      A     M      3.3;
      =     L      0.0;
      A     L      0.0;
      A     I    264.2;
      AN    I    264.3;
      =     M   2102.2;
      A     L      0.0;
      AN    I    264.2;
      A     I    264.3;
      =     M   2102.3;
NETWORK
TITLE =

      A     M      3.3;
      =     L      0.0;
      A     L      0.0;
      A     I    264.4;
      AN    I    264.5;
      =     M   2102.4;
      A     L      0.0;
      AN    I    264.4;
      A     I    264.5;
      =     M   2102.5;
NETWORK
TITLE =
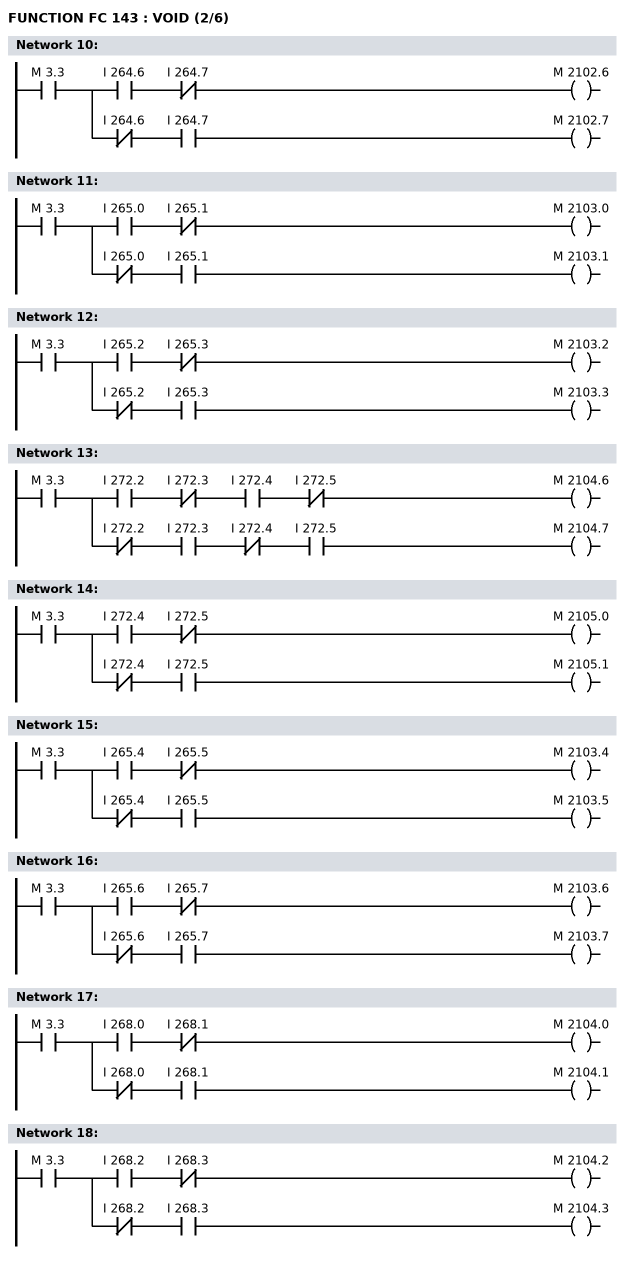

      A     M      3.3;
      =     L      0.0;
      A     L      0.0;
      A     I    264.6;
      AN    I    264.7;
      =     M   2102.6;
      A     L      0.0;
      AN    I    264.6;
      A     I    264.7;
      =     M   2102.7;
NETWORK
TITLE =

      A     M      3.3;
      =     L      0.0;
      A     L      0.0;
      A     I    265.0;
      AN    I    265.1;
      =     M   2103.0;
      A     L      0.0;
      AN    I    265.0;
      A     I    265.1;
      =     M   2103.1;
NETWORK
TITLE =

      A     M      3.3;
      =     L      0.0;
      A     L      0.0;
      A     I    265.2;
      AN    I    265.3;
      =     M   2103.2;
      A     L      0.0;
      AN    I    265.2;
      A     I    265.3;
      =     M   2103.3;
NETWORK
TITLE =

      A     M      3.3;
      =     L      0.0;
      A     L      0.0;
      A     I    272.2;
      AN    I    272.3;
      A     I    272.4;
      AN    I    272.5;
      =     M   2104.6;
      A     L      0.0;
      AN    I    272.2;
      A     I    272.3;
      AN    I    272.4;
      A     I    272.5;
      =     M   2104.7;
NETWORK
TITLE =

      A     M      3.3;
      =     L      0.0;
      A     L      0.0;
      A     I    272.4;
      AN    I    272.5;
      =     M   2105.0;
      A     L      0.0;
      AN    I    272.4;
      A     I    272.5;
      =     M   2105.1;
NETWORK
TITLE =

      A     M      3.3;
      =     L      0.0;
      A     L      0.0;
      A     I    265.4;
      AN    I    265.5;
      =     M   2103.4;
      A     L      0.0;
      AN    I    265.4;
      A     I    265.5;
      =     M   2103.5;
NETWORK
TITLE =

      A     M      3.3;
      =     L      0.0;
      A     L      0.0;
      A     I    265.6;
      AN    I    265.7;
      =     M   2103.6;
      A     L      0.0;
      AN    I    265.6;
      A     I    265.7;
      =     M   2103.7;
NETWORK
TITLE =

      A     M      3.3;
      =     L      0.0;
      A     L      0.0;
      A     I    268.0;
      AN    I    268.1;
      =     M   2104.0;
      A     L      0.0;
      AN    I    268.0;
      A     I    268.1;
      =     M   2104.1;
NETWORK
TITLE =

      A     M      3.3;
      =     L      0.0;
      A     L      0.0;
      A     I    268.2;
      AN    I    268.3;
      =     M   2104.2;
      A     L      0.0;
      AN    I    268.2;
      A     I    268.3;
      =     M   2104.3;
NETWORK
TITLE =
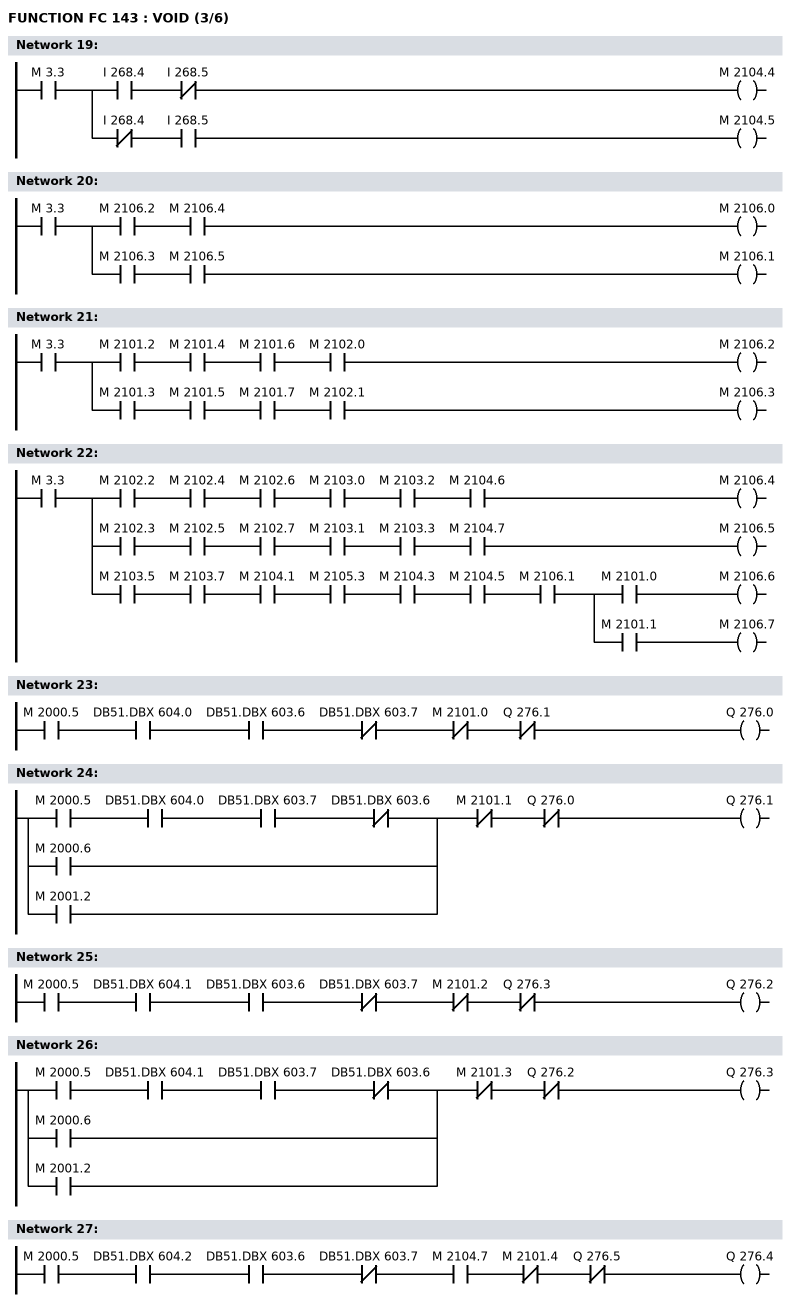

      A     M      3.3;
      =     L      0.0;
      A     L      0.0;
      A     I    268.4;
      AN    I    268.5;
      =     M   2104.4;
      A     L      0.0;
      AN    I    268.4;
      A     I    268.5;
      =     M   2104.5;
NETWORK
TITLE =

      A     M      3.3;
      =     L      0.0;
      A     L      0.0;
      A     M   2106.2;
      A     M   2106.4;
      =     M   2106.0;
      A     L      0.0;
      A     M   2106.3;
      A     M   2106.5;
      =     M   2106.1;
NETWORK
TITLE =

      A     M      3.3;
      =     L      0.0;
      A     L      0.0;
      A     M   2101.2;
      A     M   2101.4;
      A     M   2101.6;
      A     M   2102.0;
      =     M   2106.2;
      A     L      0.0;
      A     M   2101.3;
      A     M   2101.5;
      A     M   2101.7;
      A     M   2102.1;
      =     M   2106.3;
NETWORK
TITLE =

      A     M      3.3;
      =     L      0.0;
      A     L      0.0;
      A     M   2102.2;
      A     M   2102.4;
      A     M   2102.6;
      A     M   2103.0;
      A     M   2103.2;
      A     M   2104.6;
      =     M   2106.4;
      A     L      0.0;
      A     M   2102.3;
      A     M   2102.5;
      A     M   2102.7;
      A     M   2103.1;
      A     M   2103.3;
      A     M   2104.7;
      =     M   2106.5;
      A     L      0.0;
      A     M   2103.5;
      A     M   2103.7;
      A     M   2104.1;
      A     M   2105.3;
      A     M   2104.3;
      A     M   2104.5;
      A     M   2106.1;
      =     L      0.1;
      A     L      0.1;
      A     M   2101.0;
      =     M   2106.6;
      A     L      0.1;
      A     M   2101.1;
      =     M   2106.7;
NETWORK
TITLE =

      A     M   2000.5;
      A     DB51.DBX  604.0;
      A     DB51.DBX  603.6;
      AN    DB51.DBX  603.7;
      AN    M   2101.0;
      AN    Q    276.1;
      =     Q    276.0;
NETWORK
TITLE =

      A(    ;
      A     M   2000.5;
      A     DB51.DBX  604.0;
      A     DB51.DBX  603.7;
      AN    DB51.DBX  603.6;
      O     M   2000.6;
      O     M   2001.2;
      )     ;
      AN    M   2101.1;
      AN    Q    276.0;
      =     Q    276.1;
NETWORK
TITLE =

      A     M   2000.5;
      A     DB51.DBX  604.1;
      A     DB51.DBX  603.6;
      AN    DB51.DBX  603.7;
      AN    M   2101.2;
      AN    Q    276.3;
      =     Q    276.2;
NETWORK
TITLE =

      A(    ;
      A     M   2000.5;
      A     DB51.DBX  604.1;
      A     DB51.DBX  603.7;
      AN    DB51.DBX  603.6;
      O     M   2000.6;
      O     M   2001.2;
      )     ;
      AN    M   2101.3;
      AN    Q    276.2;
      =     Q    276.3;
NETWORK
TITLE =

      A     M   2000.5;
      A     DB51.DBX  604.2;
      A     DB51.DBX  603.6;
      AN    DB51.DBX  603.7;
      A     M   2104.7;
      AN    M   2101.4;
      AN    Q    276.5;
      =     Q    276.4;
NETWORK
TITLE =
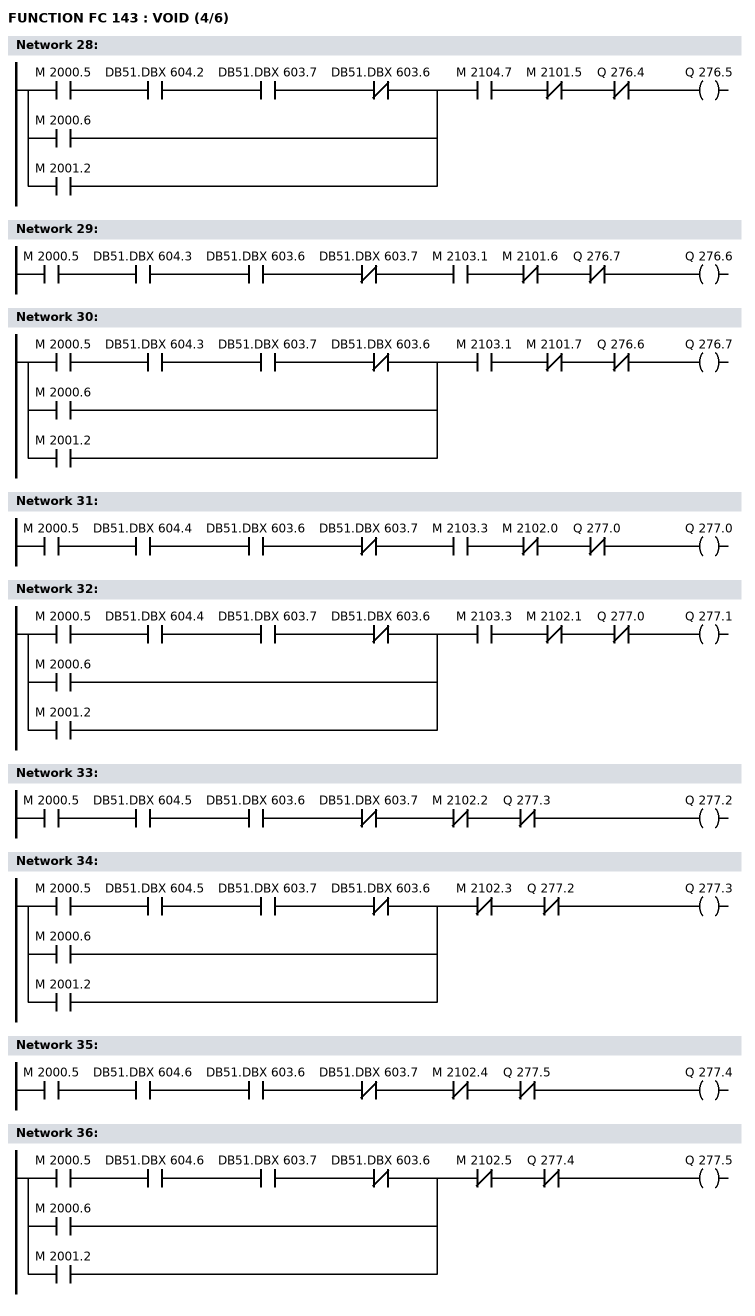

      A(    ;
      A     M   2000.5;
      A     DB51.DBX  604.2;
      A     DB51.DBX  603.7;
      AN    DB51.DBX  603.6;
      O     M   2000.6;
      O     M   2001.2;
      )     ;
      A     M   2104.7;
      AN    M   2101.5;
      AN    Q    276.4;
      =     Q    276.5;
NETWORK
TITLE =

      A     M   2000.5;
      A     DB51.DBX  604.3;
      A     DB51.DBX  603.6;
      AN    DB51.DBX  603.7;
      A     M   2103.1;
      AN    M   2101.6;
      AN    Q    276.7;
      =     Q    276.6;
NETWORK
TITLE =

      A(    ;
      A     M   2000.5;
      A     DB51.DBX  604.3;
      A     DB51.DBX  603.7;
      AN    DB51.DBX  603.6;
      O     M   2000.6;
      O     M   2001.2;
      )     ;
      A     M   2103.1;
      AN    M   2101.7;
      AN    Q    276.6;
      =     Q    276.7;
NETWORK
TITLE =

      A     M   2000.5;
      A     DB51.DBX  604.4;
      A     DB51.DBX  603.6;
      AN    DB51.DBX  603.7;
      A     M   2103.3;
      AN    M   2102.0;
      AN    Q    277.0;
      =     Q    277.0;
NETWORK
TITLE =

      A(    ;
      A     M   2000.5;
      A     DB51.DBX  604.4;
      A     DB51.DBX  603.7;
      AN    DB51.DBX  603.6;
      O     M   2000.6;
      O     M   2001.2;
      )     ;
      A     M   2103.3;
      AN    M   2102.1;
      AN    Q    277.0;
      =     Q    277.1;
NETWORK
TITLE =

      A     M   2000.5;
      A     DB51.DBX  604.5;
      A     DB51.DBX  603.6;
      AN    DB51.DBX  603.7;
      AN    M   2102.2;
      AN    Q    277.3;
      =     Q    277.2;
NETWORK
TITLE =

      A(    ;
      A     M   2000.5;
      A     DB51.DBX  604.5;
      A     DB51.DBX  603.7;
      AN    DB51.DBX  603.6;
      O     M   2000.6;
      O     M   2001.2;
      )     ;
      AN    M   2102.3;
      AN    Q    277.2;
      =     Q    277.3;
NETWORK
TITLE =

      A     M   2000.5;
      A     DB51.DBX  604.6;
      A     DB51.DBX  603.6;
      AN    DB51.DBX  603.7;
      AN    M   2102.4;
      AN    Q    277.5;
      =     Q    277.4;
NETWORK
TITLE =

      A(    ;
      A     M   2000.5;
      A     DB51.DBX  604.6;
      A     DB51.DBX  603.7;
      AN    DB51.DBX  603.6;
      O     M   2000.6;
      O     M   2001.2;
      )     ;
      AN    M   2102.5;
      AN    Q    277.4;
      =     Q    277.5;
NETWORK
TITLE =
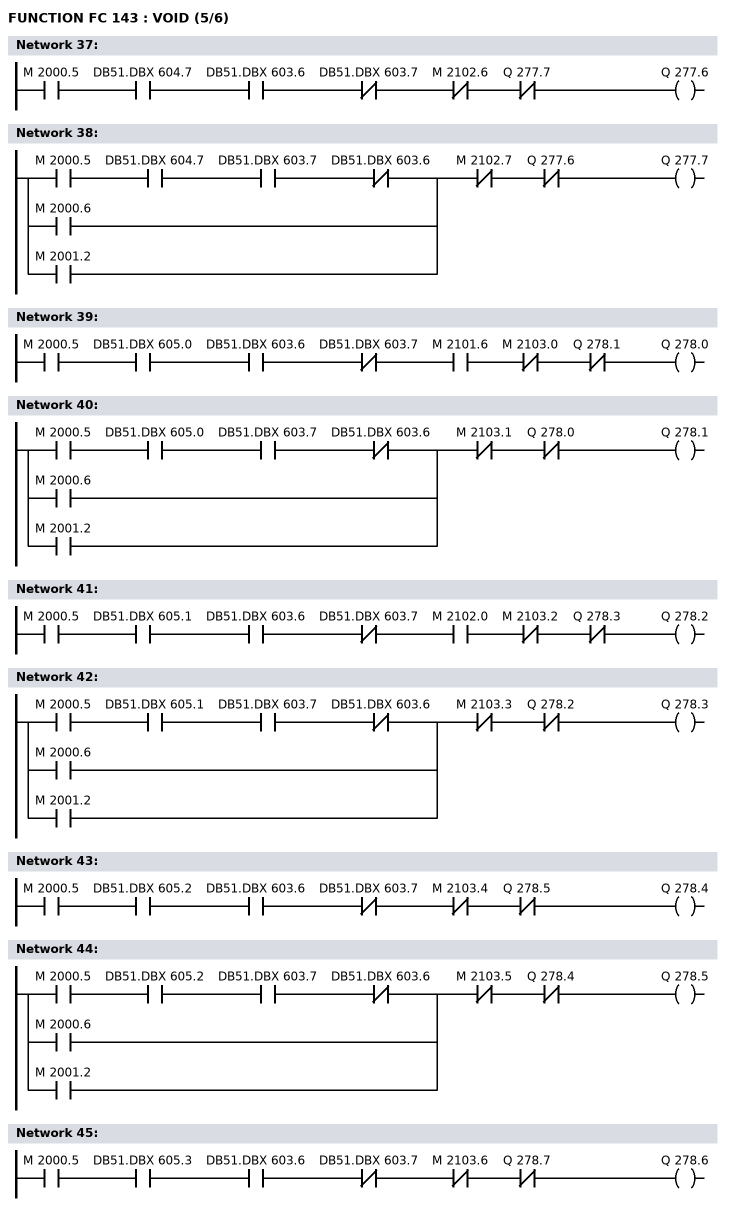

      A     M   2000.5;
      A     DB51.DBX  604.7;
      A     DB51.DBX  603.6;
      AN    DB51.DBX  603.7;
      AN    M   2102.6;
      AN    Q    277.7;
      =     Q    277.6;
NETWORK
TITLE =

      A(    ;
      A     M   2000.5;
      A     DB51.DBX  604.7;
      A     DB51.DBX  603.7;
      AN    DB51.DBX  603.6;
      O     M   2000.6;
      O     M   2001.2;
      )     ;
      AN    M   2102.7;
      AN    Q    277.6;
      =     Q    277.7;
NETWORK
TITLE =

      A     M   2000.5;
      A     DB51.DBX  605.0;
      A     DB51.DBX  603.6;
      AN    DB51.DBX  603.7;
      A     M   2101.6;
      AN    M   2103.0;
      AN    Q    278.1;
      =     Q    278.0;
NETWORK
TITLE =

      A(    ;
      A     M   2000.5;
      A     DB51.DBX  605.0;
      A     DB51.DBX  603.7;
      AN    DB51.DBX  603.6;
      O     M   2000.6;
      O     M   2001.2;
      )     ;
      AN    M   2103.1;
      AN    Q    278.0;
      =     Q    278.1;
NETWORK
TITLE =

      A     M   2000.5;
      A     DB51.DBX  605.1;
      A     DB51.DBX  603.6;
      AN    DB51.DBX  603.7;
      A     M   2102.0;
      AN    M   2103.2;
      AN    Q    278.3;
      =     Q    278.2;
NETWORK
TITLE =

      A(    ;
      A     M   2000.5;
      A     DB51.DBX  605.1;
      A     DB51.DBX  603.7;
      AN    DB51.DBX  603.6;
      O     M   2000.6;
      O     M   2001.2;
      )     ;
      AN    M   2103.3;
      AN    Q    278.2;
      =     Q    278.3;
NETWORK
TITLE =

      A     M   2000.5;
      A     DB51.DBX  605.2;
      A     DB51.DBX  603.6;
      AN    DB51.DBX  603.7;
      AN    M   2103.4;
      AN    Q    278.5;
      =     Q    278.4;
NETWORK
TITLE =

      A(    ;
      A     M   2000.5;
      A     DB51.DBX  605.2;
      A     DB51.DBX  603.7;
      AN    DB51.DBX  603.6;
      O     M   2000.6;
      O     M   2001.2;
      )     ;
      AN    M   2103.5;
      AN    Q    278.4;
      =     Q    278.5;
NETWORK
TITLE =

      A     M   2000.5;
      A     DB51.DBX  605.3;
      A     DB51.DBX  603.6;
      AN    DB51.DBX  603.7;
      AN    M   2103.6;
      AN    Q    278.7;
      =     Q    278.6;
NETWORK
TITLE =
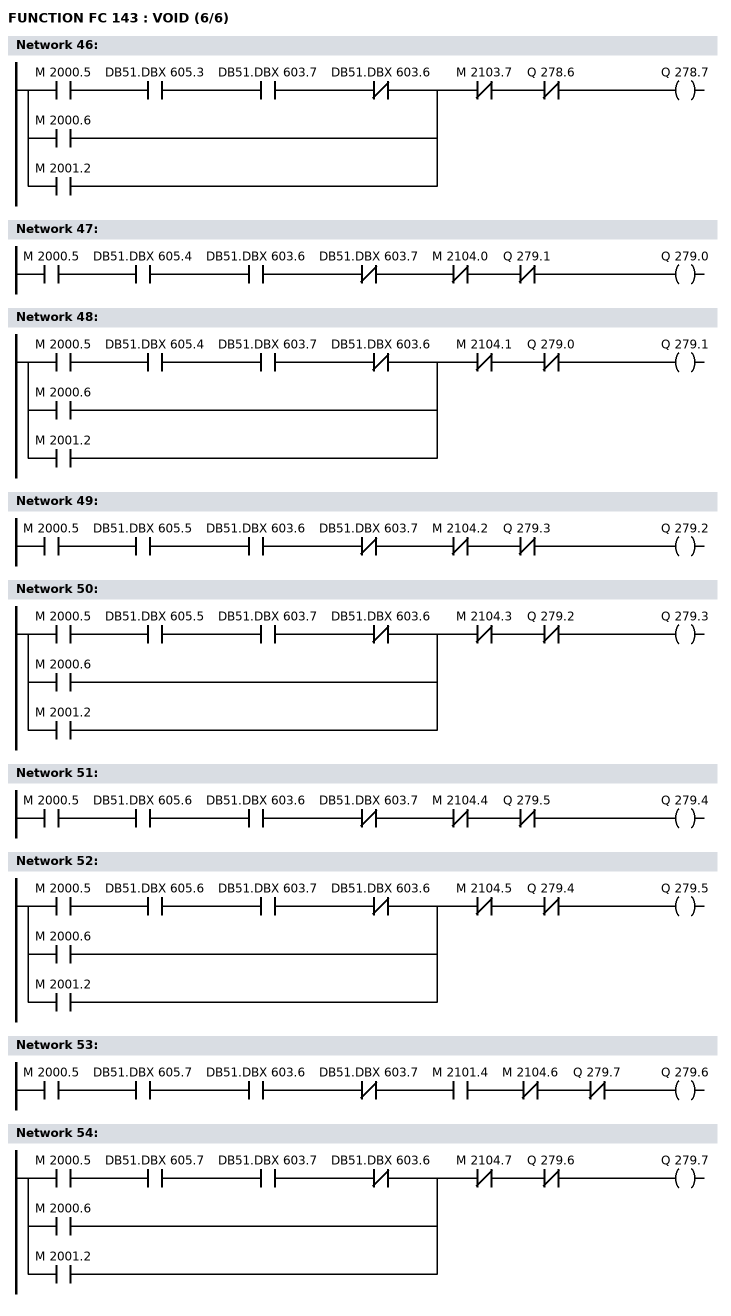

      A(    ;
      A     M   2000.5;
      A     DB51.DBX  605.3;
      A     DB51.DBX  603.7;
      AN    DB51.DBX  603.6;
      O     M   2000.6;
      O     M   2001.2;
      )     ;
      AN    M   2103.7;
      AN    Q    278.6;
      =     Q    278.7;
NETWORK
TITLE =

      A     M   2000.5;
      A     DB51.DBX  605.4;
      A     DB51.DBX  603.6;
      AN    DB51.DBX  603.7;
      AN    M   2104.0;
      AN    Q    279.1;
      =     Q    279.0;
NETWORK
TITLE =

      A(    ;
      A     M   2000.5;
      A     DB51.DBX  605.4;
      A     DB51.DBX  603.7;
      AN    DB51.DBX  603.6;
      O     M   2000.6;
      O     M   2001.2;
      )     ;
      AN    M   2104.1;
      AN    Q    279.0;
      =     Q    279.1;
NETWORK
TITLE =

      A     M   2000.5;
      A     DB51.DBX  605.5;
      A     DB51.DBX  603.6;
      AN    DB51.DBX  603.7;
      AN    M   2104.2;
      AN    Q    279.3;
      =     Q    279.2;
NETWORK
TITLE =

      A(    ;
      A     M   2000.5;
      A     DB51.DBX  605.5;
      A     DB51.DBX  603.7;
      AN    DB51.DBX  603.6;
      O     M   2000.6;
      O     M   2001.2;
      )     ;
      AN    M   2104.3;
      AN    Q    279.2;
      =     Q    279.3;
NETWORK
TITLE =

      A     M   2000.5;
      A     DB51.DBX  605.6;
      A     DB51.DBX  603.6;
      AN    DB51.DBX  603.7;
      AN    M   2104.4;
      AN    Q    279.5;
      =     Q    279.4;
NETWORK
TITLE =

      A(    ;
      A     M   2000.5;
      A     DB51.DBX  605.6;
      A     DB51.DBX  603.7;
      AN    DB51.DBX  603.6;
      O     M   2000.6;
      O     M   2001.2;
      )     ;
      AN    M   2104.5;
      AN    Q    279.4;
      =     Q    279.5;
NETWORK
TITLE =

      A     M   2000.5;
      A     DB51.DBX  605.7;
      A     DB51.DBX  603.6;
      AN    DB51.DBX  603.7;
      A     M   2101.4;
      AN    M   2104.6;
      AN    Q    279.7;
      =     Q    279.6;
NETWORK
TITLE =

      A(    ;
      A     M   2000.5;
      A     DB51.DBX  605.7;
      A     DB51.DBX  603.7;
      AN    DB51.DBX  603.6;
      O     M   2000.6;
      O     M   2001.2;
      )     ;
      AN    M   2104.7;
      AN    Q    279.6;
      =     Q    279.7;
END_FUNCTION

FUNCTION_BLOCK FB 144
TITLE =
VERSION : 0.1


VAR
  S708_TL_DC_PIN : FB 426;
  S708_TL_DC_LATCH1 : FB 426;
  S708_TL_DC_LATCH2 : FB 426;
  S708_TL_DC_1ST_CLAMP1 : FB 426;
  S708_TL_DC_1ST_CLAMP2 : FB 426;
  S708_TL_DC_1ST_CLAMP3 : FB 426;
  S708_TL_DC_2ND_CLAMP1 : FB 426;
  S708_TL_DC_2ND_CLAMP2 : FB 426;
  S708_TL_DC_U261 : FB 426;
  S708_TL_DC_U261_CLAMP : FB 426;
  S708_TL_DC_U269 : FB 426;
  S708_TL_DC_U269_CLAMP : FB 426;
  S708_TL_DC_3RD_CLAMP : FB 426;
  S708_TL_DC_U262_1_UP_DN : FB 426;
  S708_TL_DC_U262_1 : FB 426;
  S708_TL_DC_U262_1_CLAMP : FB 426;
  S708_TL_DC_U261_2_CLAMP : FB 426;
END_VAR
BEGIN
NETWORK
TITLE =
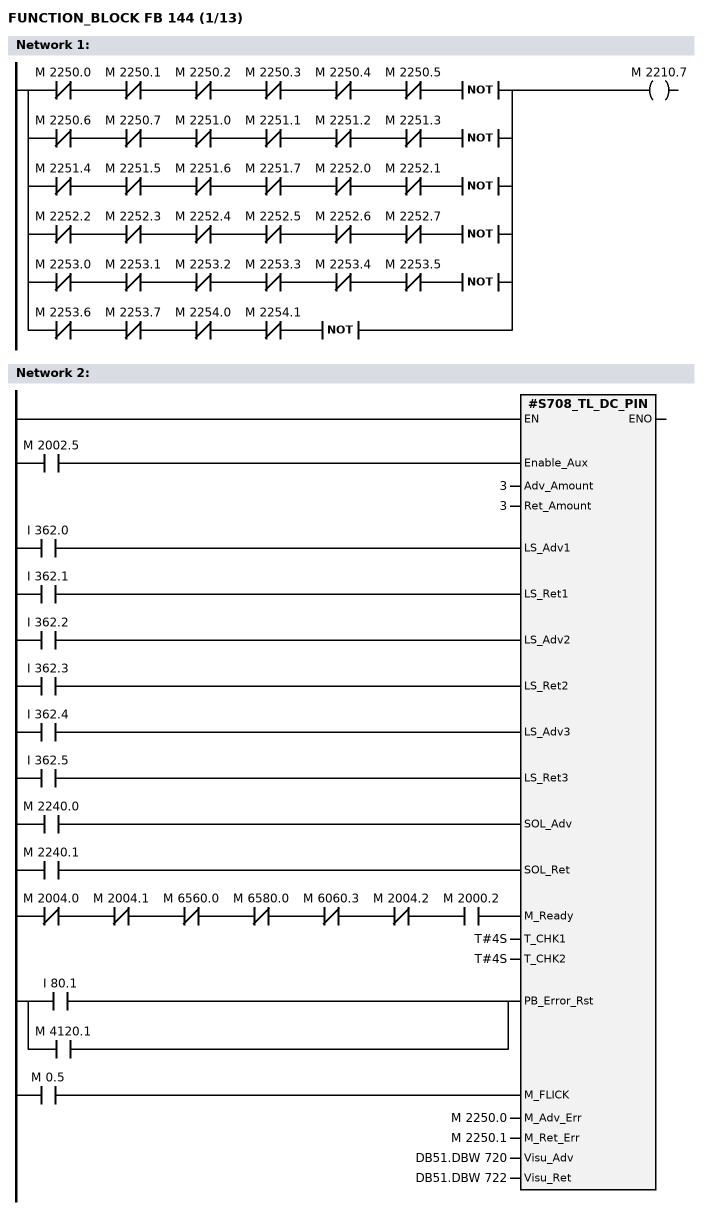

      AN    M   2250.0;
      AN    M   2250.1;
      AN    M   2250.2;
      AN    M   2250.3;
      AN    M   2250.4;
      AN    M   2250.5;
      NOT   ;
      O(    ;
      AN    M   2250.6;
      AN    M   2250.7;
      AN    M   2251.0;
      AN    M   2251.1;
      AN    M   2251.2;
      AN    M   2251.3;
      NOT   ;
      )     ;
      O(    ;
      AN    M   2251.4;
      AN    M   2251.5;
      AN    M   2251.6;
      AN    M   2251.7;
      AN    M   2252.0;
      AN    M   2252.1;
      NOT   ;
      )     ;
      O(    ;
      AN    M   2252.2;
      AN    M   2252.3;
      AN    M   2252.4;
      AN    M   2252.5;
      AN    M   2252.6;
      AN    M   2252.7;
      NOT   ;
      )     ;
      O(    ;
      AN    M   2253.0;
      AN    M   2253.1;
      AN    M   2253.2;
      AN    M   2253.3;
      AN    M   2253.4;
      AN    M   2253.5;
      NOT   ;
      )     ;
      O(    ;
      AN    M   2253.6;
      AN    M   2253.7;
      AN    M   2254.0;
      AN    M   2254.1;
      NOT   ;
      )     ;
      =     M   2210.7;
NETWORK
TITLE =

      A     M   2002.5;
      =     L      0.0;
      BLD   103;
      A     I    362.0;
      =     L      0.1;
      BLD   103;
      A     I    362.1;
      =     L      0.2;
      BLD   103;
      A     I    362.2;
      =     L      0.3;
      BLD   103;
      A     I    362.3;
      =     L      0.4;
      BLD   103;
      A     I    362.4;
      =     L      0.5;
      BLD   103;
      A     I    362.5;
      =     L      0.6;
      BLD   103;
      A     M   2240.0;
      =     L      2.1;
      BLD   103;
      A     M   2240.1;
      =     L      2.2;
      BLD   103;
      AN    M   2004.0;
      AN    M   2004.1;
      AN    M   6560.0;
      AN    M   6580.0;
      AN    M   6060.3;
      AN    M   2004.2;
      A     M   2000.2;
      =     L      2.3;
      BLD   103;
      A(    ;
      O     I     80.1;
      O     M   4120.1;
      )     ;
      =     L      2.5;
      BLD   103;
      A     M      0.5;
      =     L      2.6;
      BLD   103;
      CALL #S708_TL_DC_PIN (
           Enable_Aux               := L      0.0,
           Adv_Amount               := 3,
           Ret_Amount               := 3,
           LS_Adv1                  := L      0.1,
           LS_Ret1                  := L      0.2,
           LS_Adv2                  := L      0.3,
           LS_Ret2                  := L      0.4,
           LS_Adv3                  := L      0.5,
           LS_Ret3                  := L      0.6,
           SOL_Adv                  := L      2.1,
           SOL_Ret                  := L      2.2,
           M_Ready                  := L      2.3,
           T_CHK1                   := T#4S,
           T_CHK2                   := T#4S,
           PB_Error_Rst             := L      2.5,
           M_FLICK                  := L      2.6,
           M_Adv_Err                := M   2250.0,
           M_Ret_Err                := M   2250.1,
           Visu_Adv                 := DB51.DBW  720,
           Visu_Ret                 := DB51.DBW  722);
      NOP   0;
NETWORK
TITLE =
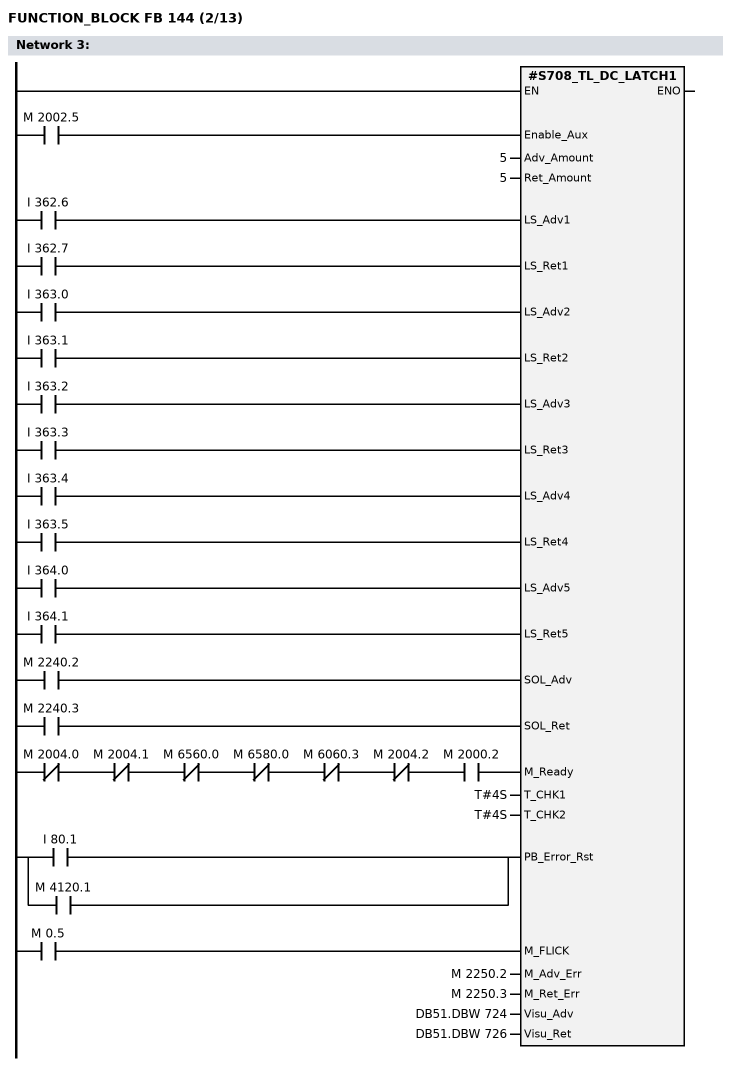

      A     M   2002.5;
      =     L      0.0;
      BLD   103;
      A     I    362.6;
      =     L      0.1;
      BLD   103;
      A     I    362.7;
      =     L      0.2;
      BLD   103;
      A     I    363.0;
      =     L      0.3;
      BLD   103;
      A     I    363.1;
      =     L      0.4;
      BLD   103;
      A     I    363.2;
      =     L      0.5;
      BLD   103;
      A     I    363.3;
      =     L      0.6;
      BLD   103;
      A     I    363.4;
      =     L      0.7;
      BLD   103;
      A     I    363.5;
      =     L      1.0;
      BLD   103;
      A     I    364.0;
      =     L      1.1;
      BLD   103;
      A     I    364.1;
      =     L      1.2;
      BLD   103;
      A     M   2240.2;
      =     L      2.1;
      BLD   103;
      A     M   2240.3;
      =     L      2.2;
      BLD   103;
      AN    M   2004.0;
      AN    M   2004.1;
      AN    M   6560.0;
      AN    M   6580.0;
      AN    M   6060.3;
      AN    M   2004.2;
      A     M   2000.2;
      =     L      2.3;
      BLD   103;
      A(    ;
      O     I     80.1;
      O     M   4120.1;
      )     ;
      =     L      2.5;
      BLD   103;
      A     M      0.5;
      =     L      2.6;
      BLD   103;
      CALL #S708_TL_DC_LATCH1 (
           Enable_Aux               := L      0.0,
           Adv_Amount               := 5,
           Ret_Amount               := 5,
           LS_Adv1                  := L      0.1,
           LS_Ret1                  := L      0.2,
           LS_Adv2                  := L      0.3,
           LS_Ret2                  := L      0.4,
           LS_Adv3                  := L      0.5,
           LS_Ret3                  := L      0.6,
           LS_Adv4                  := L      0.7,
           LS_Ret4                  := L      1.0,
           LS_Adv5                  := L      1.1,
           LS_Ret5                  := L      1.2,
           SOL_Adv                  := L      2.1,
           SOL_Ret                  := L      2.2,
           M_Ready                  := L      2.3,
           T_CHK1                   := T#4S,
           T_CHK2                   := T#4S,
           PB_Error_Rst             := L      2.5,
           M_FLICK                  := L      2.6,
           M_Adv_Err                := M   2250.2,
           M_Ret_Err                := M   2250.3,
           Visu_Adv                 := DB51.DBW  724,
           Visu_Ret                 := DB51.DBW  726);
      NOP   0;
NETWORK
TITLE =
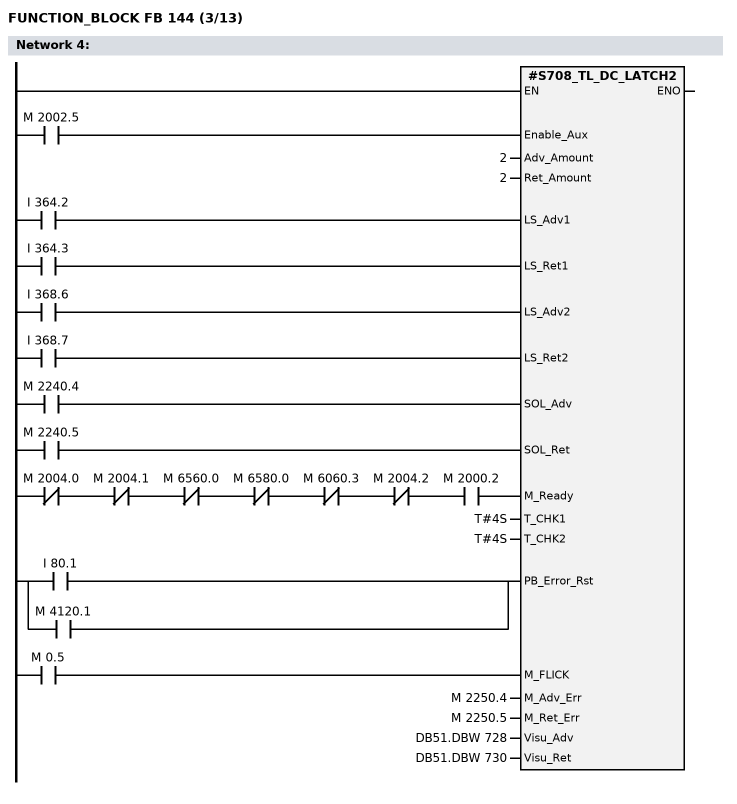

      A     M   2002.5;
      =     L      0.0;
      BLD   103;
      A     I    364.2;
      =     L      0.1;
      BLD   103;
      A     I    364.3;
      =     L      0.2;
      BLD   103;
      A     I    368.6;
      =     L      0.3;
      BLD   103;
      A     I    368.7;
      =     L      0.4;
      BLD   103;
      A     M   2240.4;
      =     L      2.1;
      BLD   103;
      A     M   2240.5;
      =     L      2.2;
      BLD   103;
      AN    M   2004.0;
      AN    M   2004.1;
      AN    M   6560.0;
      AN    M   6580.0;
      AN    M   6060.3;
      AN    M   2004.2;
      A     M   2000.2;
      =     L      2.3;
      BLD   103;
      A(    ;
      O     I     80.1;
      O     M   4120.1;
      )     ;
      =     L      2.5;
      BLD   103;
      A     M      0.5;
      =     L      2.6;
      BLD   103;
      CALL #S708_TL_DC_LATCH2 (
           Enable_Aux               := L      0.0,
           Adv_Amount               := 2,
           Ret_Amount               := 2,
           LS_Adv1                  := L      0.1,
           LS_Ret1                  := L      0.2,
           LS_Adv2                  := L      0.3,
           LS_Ret2                  := L      0.4,
           SOL_Adv                  := L      2.1,
           SOL_Ret                  := L      2.2,
           M_Ready                  := L      2.3,
           T_CHK1                   := T#4S,
           T_CHK2                   := T#4S,
           PB_Error_Rst             := L      2.5,
           M_FLICK                  := L      2.6,
           M_Adv_Err                := M   2250.4,
           M_Ret_Err                := M   2250.5,
           Visu_Adv                 := DB51.DBW  728,
           Visu_Ret                 := DB51.DBW  730);
      NOP   0;
NETWORK
TITLE =
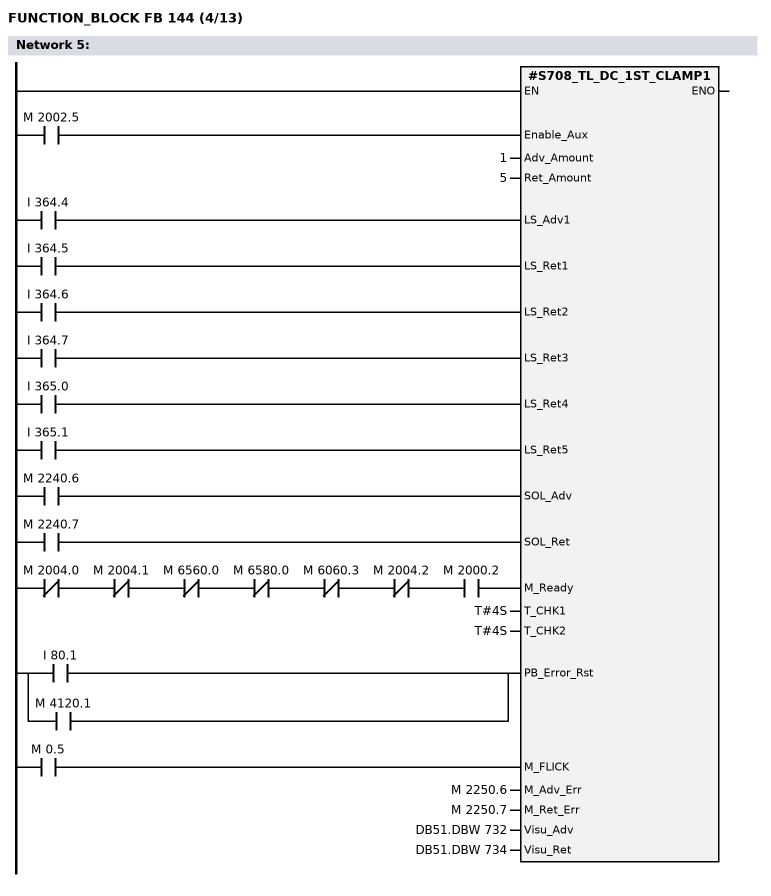

      A     M   2002.5;
      =     L      0.0;
      BLD   103;
      A     I    364.4;
      =     L      0.1;
      BLD   103;
      A     I    364.5;
      =     L      0.2;
      BLD   103;
      A     I    364.6;
      =     L      0.4;
      BLD   103;
      A     I    364.7;
      =     L      0.6;
      BLD   103;
      A     I    365.0;
      =     L      1.0;
      BLD   103;
      A     I    365.1;
      =     L      1.2;
      BLD   103;
      A     M   2240.6;
      =     L      2.1;
      BLD   103;
      A     M   2240.7;
      =     L      2.2;
      BLD   103;
      AN    M   2004.0;
      AN    M   2004.1;
      AN    M   6560.0;
      AN    M   6580.0;
      AN    M   6060.3;
      AN    M   2004.2;
      A     M   2000.2;
      =     L      2.3;
      BLD   103;
      A(    ;
      O     I     80.1;
      O     M   4120.1;
      )     ;
      =     L      2.5;
      BLD   103;
      A     M      0.5;
      =     L      2.6;
      BLD   103;
      CALL #S708_TL_DC_1ST_CLAMP1 (
           Enable_Aux               := L      0.0,
           Adv_Amount               := 1,
           Ret_Amount               := 5,
           LS_Adv1                  := L      0.1,
           LS_Ret1                  := L      0.2,
           LS_Ret2                  := L      0.4,
           LS_Ret3                  := L      0.6,
           LS_Ret4                  := L      1.0,
           LS_Ret5                  := L      1.2,
           SOL_Adv                  := L      2.1,
           SOL_Ret                  := L      2.2,
           M_Ready                  := L      2.3,
           T_CHK1                   := T#4S,
           T_CHK2                   := T#4S,
           PB_Error_Rst             := L      2.5,
           M_FLICK                  := L      2.6,
           M_Adv_Err                := M   2250.6,
           M_Ret_Err                := M   2250.7,
           Visu_Adv                 := DB51.DBW  732,
           Visu_Ret                 := DB51.DBW  734);
      NOP   0;
NETWORK
TITLE =
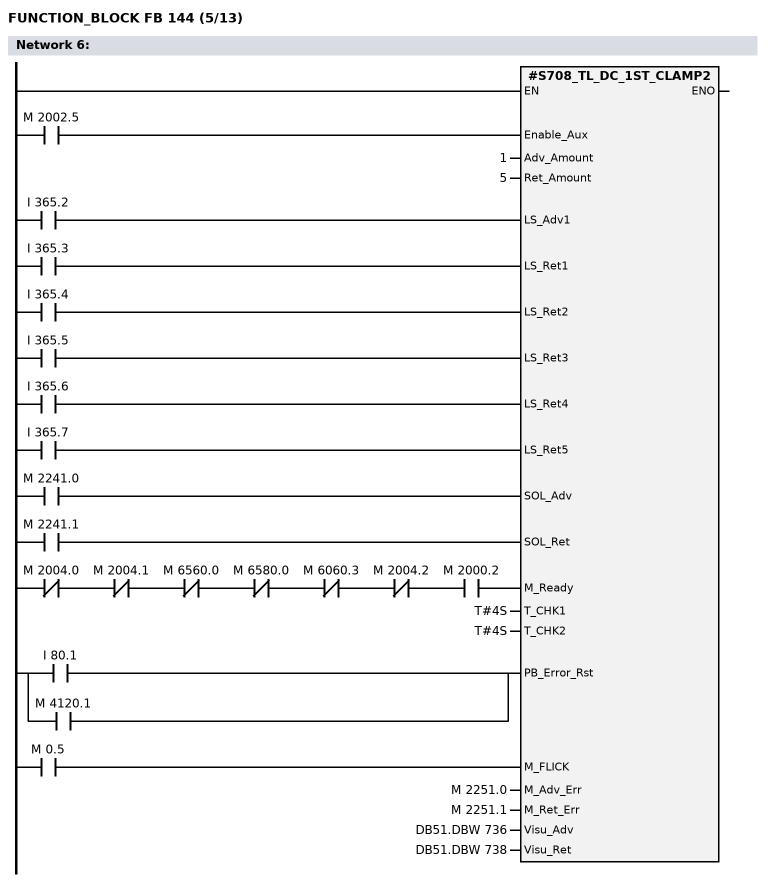

      A     M   2002.5;
      =     L      0.0;
      BLD   103;
      A     I    365.2;
      =     L      0.1;
      BLD   103;
      A     I    365.3;
      =     L      0.2;
      BLD   103;
      A     I    365.4;
      =     L      0.4;
      BLD   103;
      A     I    365.5;
      =     L      0.6;
      BLD   103;
      A     I    365.6;
      =     L      1.0;
      BLD   103;
      A     I    365.7;
      =     L      1.2;
      BLD   103;
      A     M   2241.0;
      =     L      2.1;
      BLD   103;
      A     M   2241.1;
      =     L      2.2;
      BLD   103;
      AN    M   2004.0;
      AN    M   2004.1;
      AN    M   6560.0;
      AN    M   6580.0;
      AN    M   6060.3;
      AN    M   2004.2;
      A     M   2000.2;
      =     L      2.3;
      BLD   103;
      A(    ;
      O     I     80.1;
      O     M   4120.1;
      )     ;
      =     L      2.5;
      BLD   103;
      A     M      0.5;
      =     L      2.6;
      BLD   103;
      CALL #S708_TL_DC_1ST_CLAMP2 (
           Enable_Aux               := L      0.0,
           Adv_Amount               := 1,
           Ret_Amount               := 5,
           LS_Adv1                  := L      0.1,
           LS_Ret1                  := L      0.2,
           LS_Ret2                  := L      0.4,
           LS_Ret3                  := L      0.6,
           LS_Ret4                  := L      1.0,
           LS_Ret5                  := L      1.2,
           SOL_Adv                  := L      2.1,
           SOL_Ret                  := L      2.2,
           M_Ready                  := L      2.3,
           T_CHK1                   := T#4S,
           T_CHK2                   := T#4S,
           PB_Error_Rst             := L      2.5,
           M_FLICK                  := L      2.6,
           M_Adv_Err                := M   2251.0,
           M_Ret_Err                := M   2251.1,
           Visu_Adv                 := DB51.DBW  736,
           Visu_Ret                 := DB51.DBW  738);
      NOP   0;
NETWORK
TITLE =
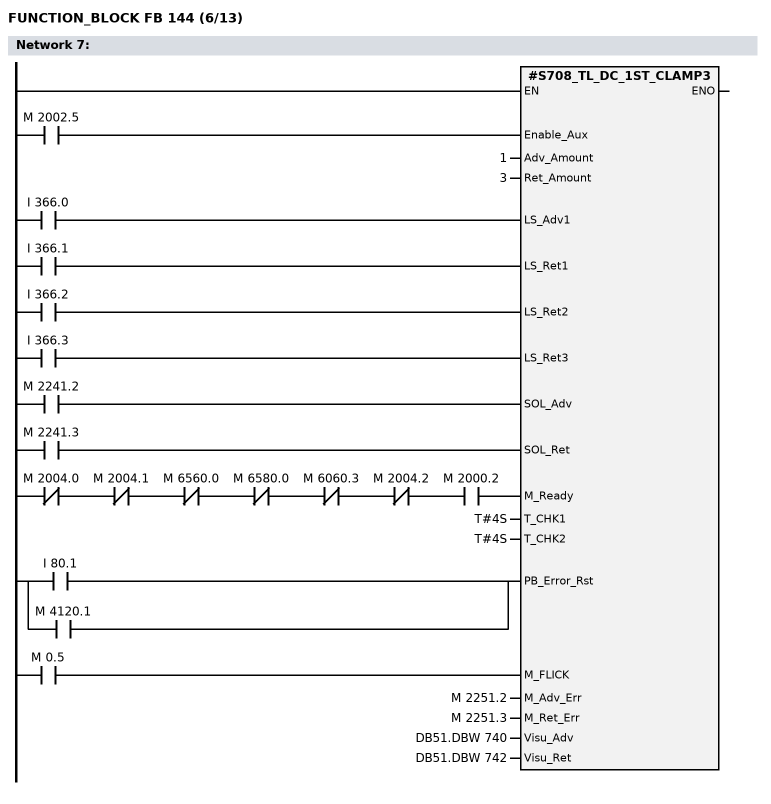

      A     M   2002.5;
      =     L      0.0;
      BLD   103;
      A     I    366.0;
      =     L      0.1;
      BLD   103;
      A     I    366.1;
      =     L      0.2;
      BLD   103;
      A     I    366.2;
      =     L      0.4;
      BLD   103;
      A     I    366.3;
      =     L      0.6;
      BLD   103;
      A     M   2241.2;
      =     L      2.1;
      BLD   103;
      A     M   2241.3;
      =     L      2.2;
      BLD   103;
      AN    M   2004.0;
      AN    M   2004.1;
      AN    M   6560.0;
      AN    M   6580.0;
      AN    M   6060.3;
      AN    M   2004.2;
      A     M   2000.2;
      =     L      2.3;
      BLD   103;
      A(    ;
      O     I     80.1;
      O     M   4120.1;
      )     ;
      =     L      2.5;
      BLD   103;
      A     M      0.5;
      =     L      2.6;
      BLD   103;
      CALL #S708_TL_DC_1ST_CLAMP3 (
           Enable_Aux               := L      0.0,
           Adv_Amount               := 1,
           Ret_Amount               := 3,
           LS_Adv1                  := L      0.1,
           LS_Ret1                  := L      0.2,
           LS_Ret2                  := L      0.4,
           LS_Ret3                  := L      0.6,
           SOL_Adv                  := L      2.1,
           SOL_Ret                  := L      2.2,
           M_Ready                  := L      2.3,
           T_CHK1                   := T#4S,
           T_CHK2                   := T#4S,
           PB_Error_Rst             := L      2.5,
           M_FLICK                  := L      2.6,
           M_Adv_Err                := M   2251.2,
           M_Ret_Err                := M   2251.3,
           Visu_Adv                 := DB51.DBW  740,
           Visu_Ret                 := DB51.DBW  742);
      NOP   0;
NETWORK
TITLE =
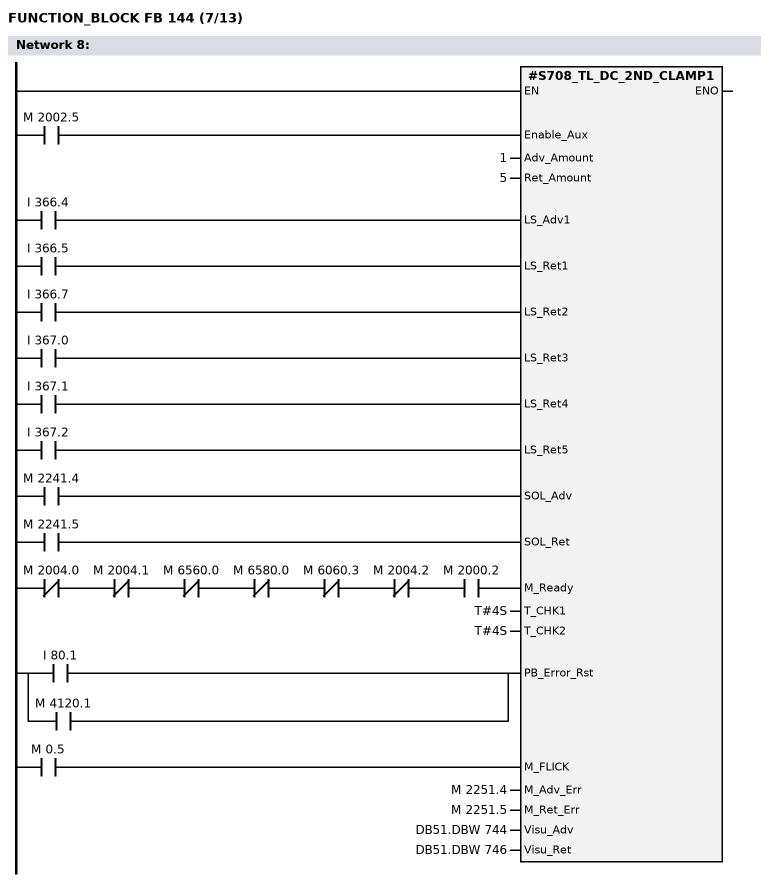

      A     M   2002.5;
      =     L      0.0;
      BLD   103;
      A     I    366.4;
      =     L      0.1;
      BLD   103;
      A     I    366.5;
      =     L      0.2;
      BLD   103;
      A     I    366.7;
      =     L      0.4;
      BLD   103;
      A     I    367.0;
      =     L      0.6;
      BLD   103;
      A     I    367.1;
      =     L      1.0;
      BLD   103;
      A     I    367.2;
      =     L      1.2;
      BLD   103;
      A     M   2241.4;
      =     L      2.1;
      BLD   103;
      A     M   2241.5;
      =     L      2.2;
      BLD   103;
      AN    M   2004.0;
      AN    M   2004.1;
      AN    M   6560.0;
      AN    M   6580.0;
      AN    M   6060.3;
      AN    M   2004.2;
      A     M   2000.2;
      =     L      2.3;
      BLD   103;
      A(    ;
      O     I     80.1;
      O     M   4120.1;
      )     ;
      =     L      2.5;
      BLD   103;
      A     M      0.5;
      =     L      2.6;
      BLD   103;
      CALL #S708_TL_DC_2ND_CLAMP1 (
           Enable_Aux               := L      0.0,
           Adv_Amount               := 1,
           Ret_Amount               := 5,
           LS_Adv1                  := L      0.1,
           LS_Ret1                  := L      0.2,
           LS_Ret2                  := L      0.4,
           LS_Ret3                  := L      0.6,
           LS_Ret4                  := L      1.0,
           LS_Ret5                  := L      1.2,
           SOL_Adv                  := L      2.1,
           SOL_Ret                  := L      2.2,
           M_Ready                  := L      2.3,
           T_CHK1                   := T#4S,
           T_CHK2                   := T#4S,
           PB_Error_Rst             := L      2.5,
           M_FLICK                  := L      2.6,
           M_Adv_Err                := M   2251.4,
           M_Ret_Err                := M   2251.5,
           Visu_Adv                 := DB51.DBW  744,
           Visu_Ret                 := DB51.DBW  746);
      NOP   0;
NETWORK
TITLE =
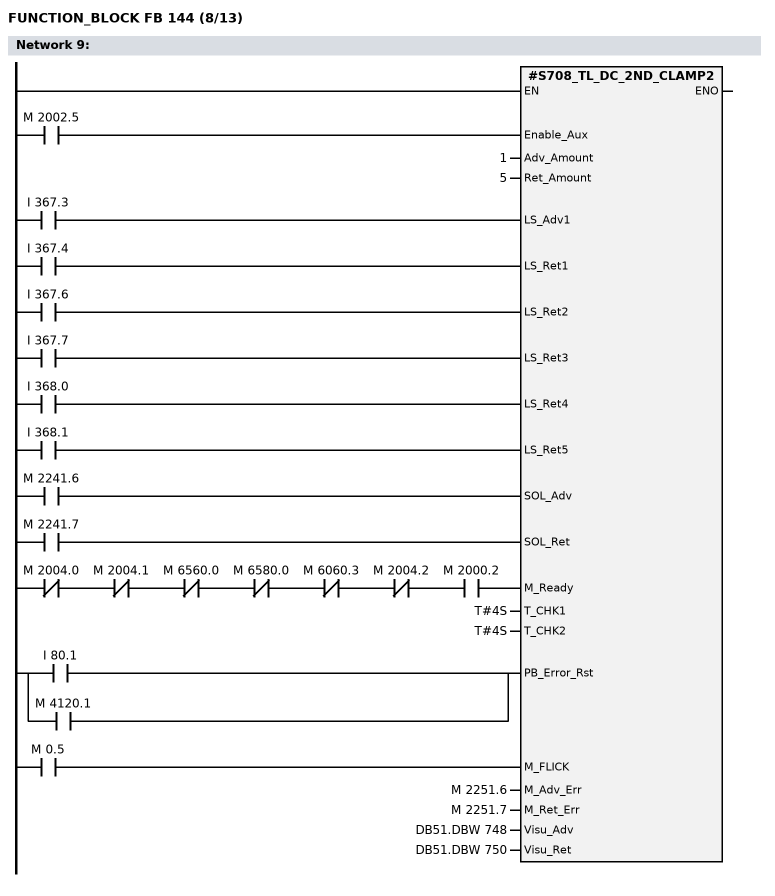

      A     M   2002.5;
      =     L      0.0;
      BLD   103;
      A     I    367.3;
      =     L      0.1;
      BLD   103;
      A     I    367.4;
      =     L      0.2;
      BLD   103;
      A     I    367.6;
      =     L      0.4;
      BLD   103;
      A     I    367.7;
      =     L      0.6;
      BLD   103;
      A     I    368.0;
      =     L      1.0;
      BLD   103;
      A     I    368.1;
      =     L      1.2;
      BLD   103;
      A     M   2241.6;
      =     L      2.1;
      BLD   103;
      A     M   2241.7;
      =     L      2.2;
      BLD   103;
      AN    M   2004.0;
      AN    M   2004.1;
      AN    M   6560.0;
      AN    M   6580.0;
      AN    M   6060.3;
      AN    M   2004.2;
      A     M   2000.2;
      =     L      2.3;
      BLD   103;
      A(    ;
      O     I     80.1;
      O     M   4120.1;
      )     ;
      =     L      2.5;
      BLD   103;
      A     M      0.5;
      =     L      2.6;
      BLD   103;
      CALL #S708_TL_DC_2ND_CLAMP2 (
           Enable_Aux               := L      0.0,
           Adv_Amount               := 1,
           Ret_Amount               := 5,
           LS_Adv1                  := L      0.1,
           LS_Ret1                  := L      0.2,
           LS_Ret2                  := L      0.4,
           LS_Ret3                  := L      0.6,
           LS_Ret4                  := L      1.0,
           LS_Ret5                  := L      1.2,
           SOL_Adv                  := L      2.1,
           SOL_Ret                  := L      2.2,
           M_Ready                  := L      2.3,
           T_CHK1                   := T#4S,
           T_CHK2                   := T#4S,
           PB_Error_Rst             := L      2.5,
           M_FLICK                  := L      2.6,
           M_Adv_Err                := M   2251.6,
           M_Ret_Err                := M   2251.7,
           Visu_Adv                 := DB51.DBW  748,
           Visu_Ret                 := DB51.DBW  750);
      NOP   0;
NETWORK
TITLE =
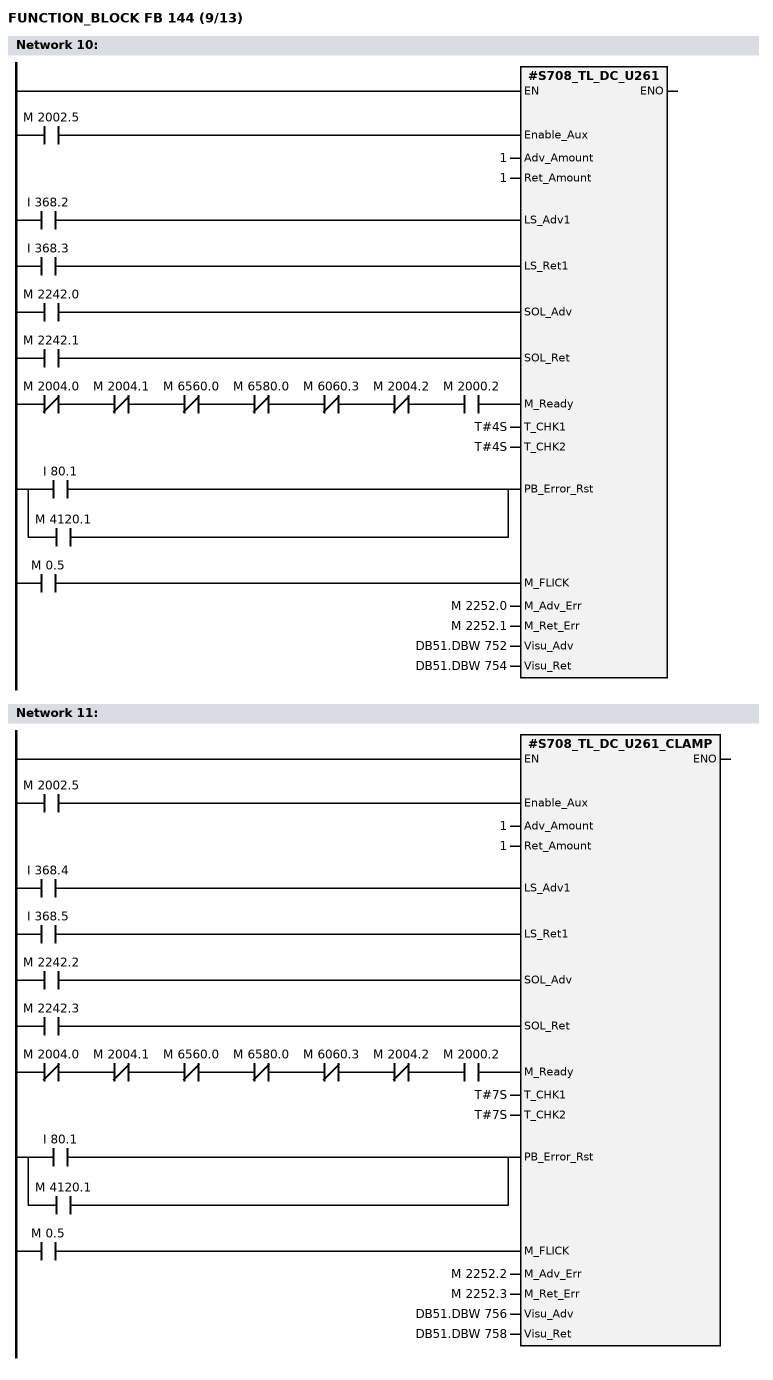

      A     M   2002.5;
      =     L      0.0;
      BLD   103;
      A     I    368.2;
      =     L      0.1;
      BLD   103;
      A     I    368.3;
      =     L      0.2;
      BLD   103;
      A     M   2242.0;
      =     L      2.1;
      BLD   103;
      A     M   2242.1;
      =     L      2.2;
      BLD   103;
      AN    M   2004.0;
      AN    M   2004.1;
      AN    M   6560.0;
      AN    M   6580.0;
      AN    M   6060.3;
      AN    M   2004.2;
      A     M   2000.2;
      =     L      2.3;
      BLD   103;
      A(    ;
      O     I     80.1;
      O     M   4120.1;
      )     ;
      =     L      2.5;
      BLD   103;
      A     M      0.5;
      =     L      2.6;
      BLD   103;
      CALL #S708_TL_DC_U261 (
           Enable_Aux               := L      0.0,
           Adv_Amount               := 1,
           Ret_Amount               := 1,
           LS_Adv1                  := L      0.1,
           LS_Ret1                  := L      0.2,
           SOL_Adv                  := L      2.1,
           SOL_Ret                  := L      2.2,
           M_Ready                  := L      2.3,
           T_CHK1                   := T#4S,
           T_CHK2                   := T#4S,
           PB_Error_Rst             := L      2.5,
           M_FLICK                  := L      2.6,
           M_Adv_Err                := M   2252.0,
           M_Ret_Err                := M   2252.1,
           Visu_Adv                 := DB51.DBW  752,
           Visu_Ret                 := DB51.DBW  754);
      NOP   0;
NETWORK
TITLE =

      A     M   2002.5;
      =     L      0.0;
      BLD   103;
      A     I    368.4;
      =     L      0.1;
      BLD   103;
      A     I    368.5;
      =     L      0.2;
      BLD   103;
      A     M   2242.2;
      =     L      2.1;
      BLD   103;
      A     M   2242.3;
      =     L      2.2;
      BLD   103;
      AN    M   2004.0;
      AN    M   2004.1;
      AN    M   6560.0;
      AN    M   6580.0;
      AN    M   6060.3;
      AN    M   2004.2;
      A     M   2000.2;
      =     L      2.3;
      BLD   103;
      A(    ;
      O     I     80.1;
      O     M   4120.1;
      )     ;
      =     L      2.5;
      BLD   103;
      A     M      0.5;
      =     L      2.6;
      BLD   103;
      CALL #S708_TL_DC_U261_CLAMP (
           Enable_Aux               := L      0.0,
           Adv_Amount               := 1,
           Ret_Amount               := 1,
           LS_Adv1                  := L      0.1,
           LS_Ret1                  := L      0.2,
           SOL_Adv                  := L      2.1,
           SOL_Ret                  := L      2.2,
           M_Ready                  := L      2.3,
           T_CHK1                   := T#7S,
           T_CHK2                   := T#7S,
           PB_Error_Rst             := L      2.5,
           M_FLICK                  := L      2.6,
           M_Adv_Err                := M   2252.2,
           M_Ret_Err                := M   2252.3,
           Visu_Adv                 := DB51.DBW  756,
           Visu_Ret                 := DB51.DBW  758);
      NOP   0;
NETWORK
TITLE =
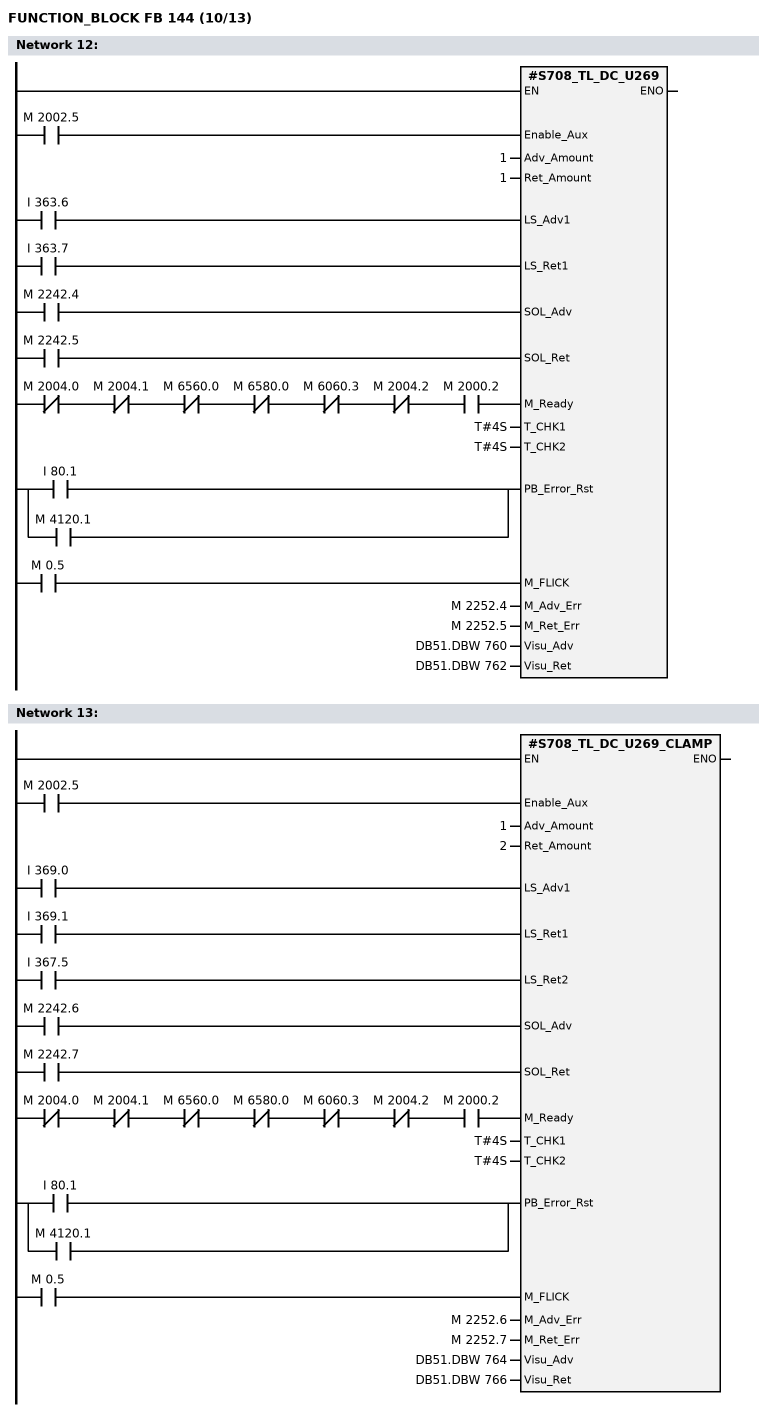

      A     M   2002.5;
      =     L      0.0;
      BLD   103;
      A     I    363.6;
      =     L      0.1;
      BLD   103;
      A     I    363.7;
      =     L      0.2;
      BLD   103;
      A     M   2242.4;
      =     L      2.1;
      BLD   103;
      A     M   2242.5;
      =     L      2.2;
      BLD   103;
      AN    M   2004.0;
      AN    M   2004.1;
      AN    M   6560.0;
      AN    M   6580.0;
      AN    M   6060.3;
      AN    M   2004.2;
      A     M   2000.2;
      =     L      2.3;
      BLD   103;
      A(    ;
      O     I     80.1;
      O     M   4120.1;
      )     ;
      =     L      2.5;
      BLD   103;
      A     M      0.5;
      =     L      2.6;
      BLD   103;
      CALL #S708_TL_DC_U269 (
           Enable_Aux               := L      0.0,
           Adv_Amount               := 1,
           Ret_Amount               := 1,
           LS_Adv1                  := L      0.1,
           LS_Ret1                  := L      0.2,
           SOL_Adv                  := L      2.1,
           SOL_Ret                  := L      2.2,
           M_Ready                  := L      2.3,
           T_CHK1                   := T#4S,
           T_CHK2                   := T#4S,
           PB_Error_Rst             := L      2.5,
           M_FLICK                  := L      2.6,
           M_Adv_Err                := M   2252.4,
           M_Ret_Err                := M   2252.5,
           Visu_Adv                 := DB51.DBW  760,
           Visu_Ret                 := DB51.DBW  762);
      NOP   0;
NETWORK
TITLE =

      A     M   2002.5;
      =     L      0.0;
      BLD   103;
      A     I    369.0;
      =     L      0.1;
      BLD   103;
      A     I    369.1;
      =     L      0.2;
      BLD   103;
      A     I    367.5;
      =     L      0.4;
      BLD   103;
      A     M   2242.6;
      =     L      2.1;
      BLD   103;
      A     M   2242.7;
      =     L      2.2;
      BLD   103;
      AN    M   2004.0;
      AN    M   2004.1;
      AN    M   6560.0;
      AN    M   6580.0;
      AN    M   6060.3;
      AN    M   2004.2;
      A     M   2000.2;
      =     L      2.3;
      BLD   103;
      A(    ;
      O     I     80.1;
      O     M   4120.1;
      )     ;
      =     L      2.5;
      BLD   103;
      A     M      0.5;
      =     L      2.6;
      BLD   103;
      CALL #S708_TL_DC_U269_CLAMP (
           Enable_Aux               := L      0.0,
           Adv_Amount               := 1,
           Ret_Amount               := 2,
           LS_Adv1                  := L      0.1,
           LS_Ret1                  := L      0.2,
           LS_Ret2                  := L      0.4,
           SOL_Adv                  := L      2.1,
           SOL_Ret                  := L      2.2,
           M_Ready                  := L      2.3,
           T_CHK1                   := T#4S,
           T_CHK2                   := T#4S,
           PB_Error_Rst             := L      2.5,
           M_FLICK                  := L      2.6,
           M_Adv_Err                := M   2252.6,
           M_Ret_Err                := M   2252.7,
           Visu_Adv                 := DB51.DBW  764,
           Visu_Ret                 := DB51.DBW  766);
      NOP   0;
NETWORK
TITLE =
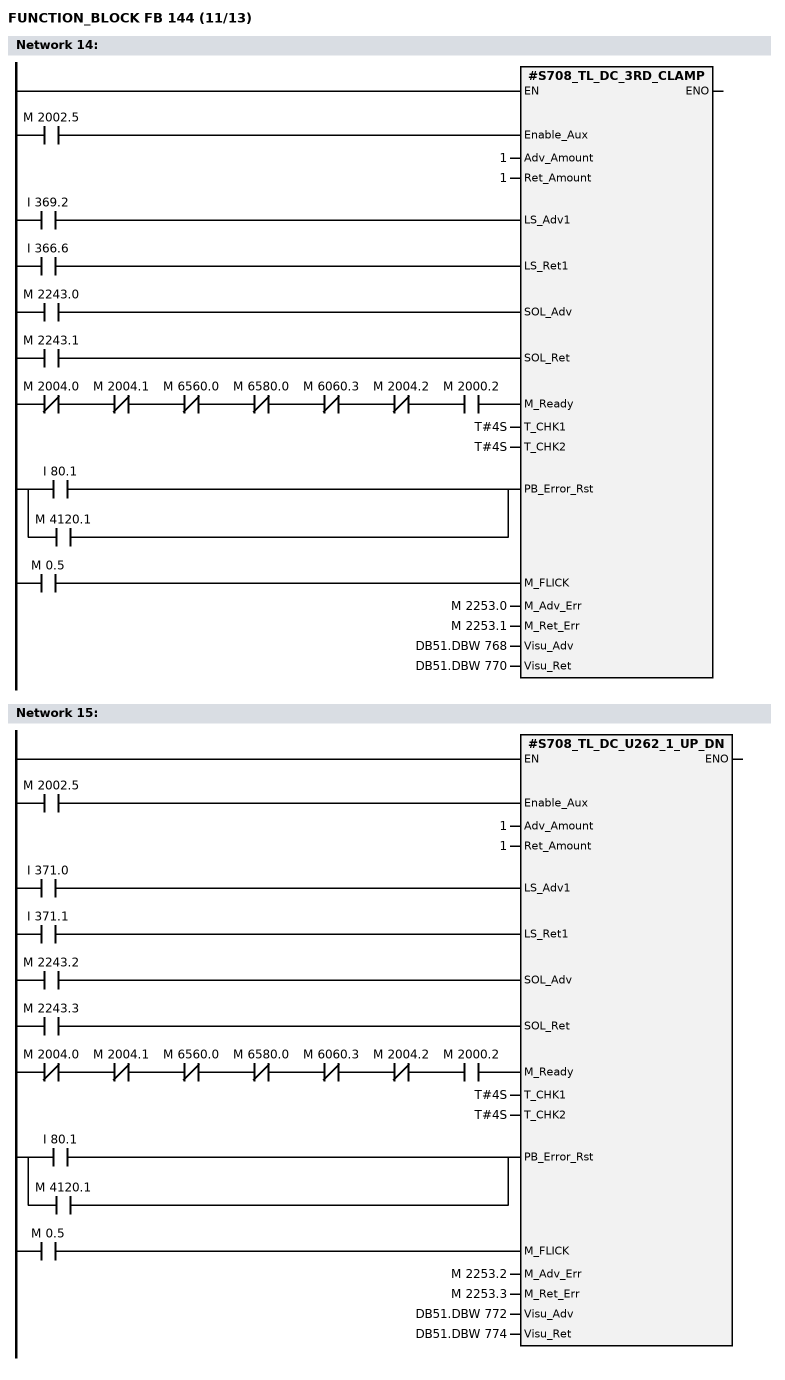

      A     M   2002.5;
      =     L      0.0;
      BLD   103;
      A     I    369.2;
      =     L      0.1;
      BLD   103;
      A     I    366.6;
      =     L      0.2;
      BLD   103;
      A     M   2243.0;
      =     L      2.1;
      BLD   103;
      A     M   2243.1;
      =     L      2.2;
      BLD   103;
      AN    M   2004.0;
      AN    M   2004.1;
      AN    M   6560.0;
      AN    M   6580.0;
      AN    M   6060.3;
      AN    M   2004.2;
      A     M   2000.2;
      =     L      2.3;
      BLD   103;
      A(    ;
      O     I     80.1;
      O     M   4120.1;
      )     ;
      =     L      2.5;
      BLD   103;
      A     M      0.5;
      =     L      2.6;
      BLD   103;
      CALL #S708_TL_DC_3RD_CLAMP (
           Enable_Aux               := L      0.0,
           Adv_Amount               := 1,
           Ret_Amount               := 1,
           LS_Adv1                  := L      0.1,
           LS_Ret1                  := L      0.2,
           SOL_Adv                  := L      2.1,
           SOL_Ret                  := L      2.2,
           M_Ready                  := L      2.3,
           T_CHK1                   := T#4S,
           T_CHK2                   := T#4S,
           PB_Error_Rst             := L      2.5,
           M_FLICK                  := L      2.6,
           M_Adv_Err                := M   2253.0,
           M_Ret_Err                := M   2253.1,
           Visu_Adv                 := DB51.DBW  768,
           Visu_Ret                 := DB51.DBW  770);
      NOP   0;
NETWORK
TITLE =

      A     M   2002.5;
      =     L      0.0;
      BLD   103;
      A     I    371.0;
      =     L      0.1;
      BLD   103;
      A     I    371.1;
      =     L      0.2;
      BLD   103;
      A     M   2243.2;
      =     L      2.1;
      BLD   103;
      A     M   2243.3;
      =     L      2.2;
      BLD   103;
      AN    M   2004.0;
      AN    M   2004.1;
      AN    M   6560.0;
      AN    M   6580.0;
      AN    M   6060.3;
      AN    M   2004.2;
      A     M   2000.2;
      =     L      2.3;
      BLD   103;
      A(    ;
      O     I     80.1;
      O     M   4120.1;
      )     ;
      =     L      2.5;
      BLD   103;
      A     M      0.5;
      =     L      2.6;
      BLD   103;
      CALL #S708_TL_DC_U262_1_UP_DN (
           Enable_Aux               := L      0.0,
           Adv_Amount               := 1,
           Ret_Amount               := 1,
           LS_Adv1                  := L      0.1,
           LS_Ret1                  := L      0.2,
           SOL_Adv                  := L      2.1,
           SOL_Ret                  := L      2.2,
           M_Ready                  := L      2.3,
           T_CHK1                   := T#4S,
           T_CHK2                   := T#4S,
           PB_Error_Rst             := L      2.5,
           M_FLICK                  := L      2.6,
           M_Adv_Err                := M   2253.2,
           M_Ret_Err                := M   2253.3,
           Visu_Adv                 := DB51.DBW  772,
           Visu_Ret                 := DB51.DBW  774);
      NOP   0;
NETWORK
TITLE =
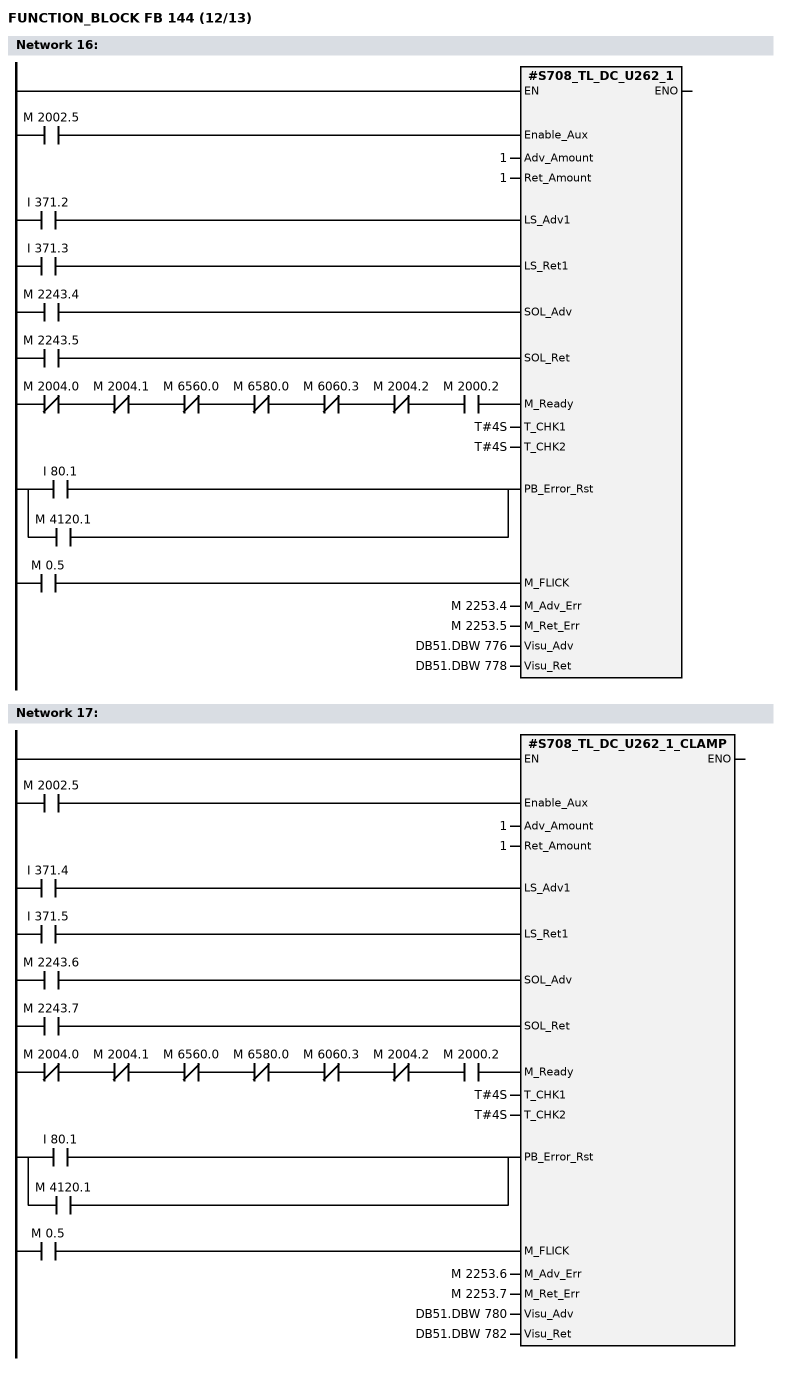

      A     M   2002.5;
      =     L      0.0;
      BLD   103;
      A     I    371.2;
      =     L      0.1;
      BLD   103;
      A     I    371.3;
      =     L      0.2;
      BLD   103;
      A     M   2243.4;
      =     L      2.1;
      BLD   103;
      A     M   2243.5;
      =     L      2.2;
      BLD   103;
      AN    M   2004.0;
      AN    M   2004.1;
      AN    M   6560.0;
      AN    M   6580.0;
      AN    M   6060.3;
      AN    M   2004.2;
      A     M   2000.2;
      =     L      2.3;
      BLD   103;
      A(    ;
      O     I     80.1;
      O     M   4120.1;
      )     ;
      =     L      2.5;
      BLD   103;
      A     M      0.5;
      =     L      2.6;
      BLD   103;
      CALL #S708_TL_DC_U262_1 (
           Enable_Aux               := L      0.0,
           Adv_Amount               := 1,
           Ret_Amount               := 1,
           LS_Adv1                  := L      0.1,
           LS_Ret1                  := L      0.2,
           SOL_Adv                  := L      2.1,
           SOL_Ret                  := L      2.2,
           M_Ready                  := L      2.3,
           T_CHK1                   := T#4S,
           T_CHK2                   := T#4S,
           PB_Error_Rst             := L      2.5,
           M_FLICK                  := L      2.6,
           M_Adv_Err                := M   2253.4,
           M_Ret_Err                := M   2253.5,
           Visu_Adv                 := DB51.DBW  776,
           Visu_Ret                 := DB51.DBW  778);
      NOP   0;
NETWORK
TITLE =

      A     M   2002.5;
      =     L      0.0;
      BLD   103;
      A     I    371.4;
      =     L      0.1;
      BLD   103;
      A     I    371.5;
      =     L      0.2;
      BLD   103;
      A     M   2243.6;
      =     L      2.1;
      BLD   103;
      A     M   2243.7;
      =     L      2.2;
      BLD   103;
      AN    M   2004.0;
      AN    M   2004.1;
      AN    M   6560.0;
      AN    M   6580.0;
      AN    M   6060.3;
      AN    M   2004.2;
      A     M   2000.2;
      =     L      2.3;
      BLD   103;
      A(    ;
      O     I     80.1;
      O     M   4120.1;
      )     ;
      =     L      2.5;
      BLD   103;
      A     M      0.5;
      =     L      2.6;
      BLD   103;
      CALL #S708_TL_DC_U262_1_CLAMP (
           Enable_Aux               := L      0.0,
           Adv_Amount               := 1,
           Ret_Amount               := 1,
           LS_Adv1                  := L      0.1,
           LS_Ret1                  := L      0.2,
           SOL_Adv                  := L      2.1,
           SOL_Ret                  := L      2.2,
           M_Ready                  := L      2.3,
           T_CHK1                   := T#4S,
           T_CHK2                   := T#4S,
           PB_Error_Rst             := L      2.5,
           M_FLICK                  := L      2.6,
           M_Adv_Err                := M   2253.6,
           M_Ret_Err                := M   2253.7,
           Visu_Adv                 := DB51.DBW  780,
           Visu_Ret                 := DB51.DBW  782);
      NOP   0;
NETWORK
TITLE =
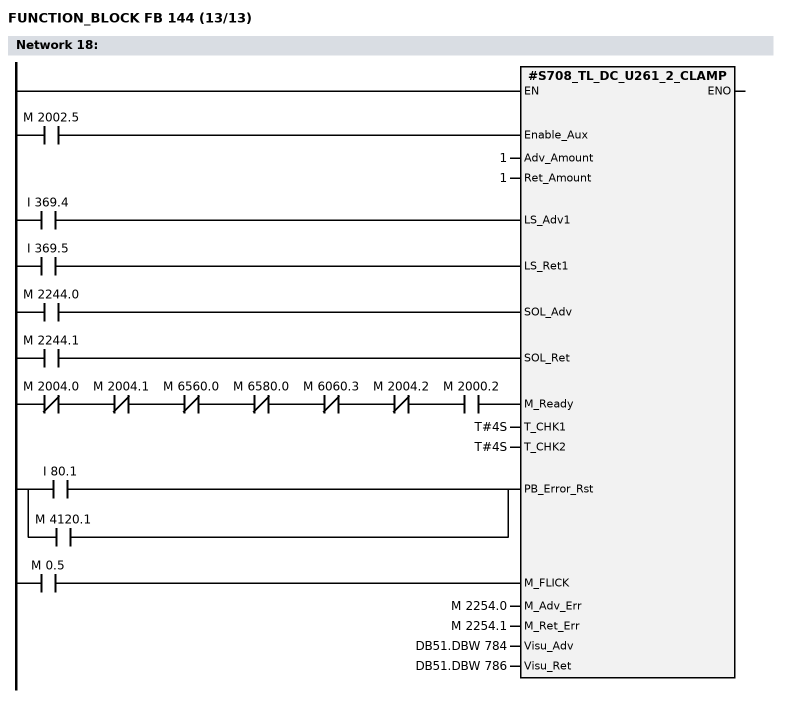

      A     M   2002.5;
      =     L      0.0;
      BLD   103;
      A     I    369.4;
      =     L      0.1;
      BLD   103;
      A     I    369.5;
      =     L      0.2;
      BLD   103;
      A     M   2244.0;
      =     L      2.1;
      BLD   103;
      A     M   2244.1;
      =     L      2.2;
      BLD   103;
      AN    M   2004.0;
      AN    M   2004.1;
      AN    M   6560.0;
      AN    M   6580.0;
      AN    M   6060.3;
      AN    M   2004.2;
      A     M   2000.2;
      =     L      2.3;
      BLD   103;
      A(    ;
      O     I     80.1;
      O     M   4120.1;
      )     ;
      =     L      2.5;
      BLD   103;
      A     M      0.5;
      =     L      2.6;
      BLD   103;
      CALL #S708_TL_DC_U261_2_CLAMP (
           Enable_Aux               := L      0.0,
           Adv_Amount               := 1,
           Ret_Amount               := 1,
           LS_Adv1                  := L      0.1,
           LS_Ret1                  := L      0.2,
           SOL_Adv                  := L      2.1,
           SOL_Ret                  := L      2.2,
           M_Ready                  := L      2.3,
           T_CHK1                   := T#4S,
           T_CHK2                   := T#4S,
           PB_Error_Rst             := L      2.5,
           M_FLICK                  := L      2.6,
           M_Adv_Err                := M   2254.0,
           M_Ret_Err                := M   2254.1,
           Visu_Adv                 := DB51.DBW  784,
           Visu_Ret                 := DB51.DBW  786);
      NOP   0;
END_FUNCTION_BLOCK

DATA_BLOCK DB 144
TITLE =
VERSION : 0.0

 FB 144
BEGIN
   S708_TL_DC_PIN.Enable_Aux := FALSE;
   S708_TL_DC_PIN.Adv_Amount := 3;
   S708_TL_DC_PIN.Ret_Amount := 3;
   S708_TL_DC_PIN.LS_Adv1 := FALSE;
   S708_TL_DC_PIN.LS_Ret1 := FALSE;
   S708_TL_DC_PIN.LS_Adv2 := FALSE;
   S708_TL_DC_PIN.LS_Ret2 := FALSE;
   S708_TL_DC_PIN.LS_Adv3 := FALSE;
   S708_TL_DC_PIN.LS_Ret3 := FALSE;
   S708_TL_DC_PIN.LS_Adv4 := FALSE;
   S708_TL_DC_PIN.LS_Ret4 := FALSE;
   S708_TL_DC_PIN.LS_Adv5 := FALSE;
   S708_TL_DC_PIN.LS_Ret5 := FALSE;
   S708_TL_DC_PIN.LS_Adv6 := FALSE;
   S708_TL_DC_PIN.LS_Ret6 := FALSE;
   S708_TL_DC_PIN.LS_Adv7 := FALSE;
   S708_TL_DC_PIN.LS_Ret7 := FALSE;
   S708_TL_DC_PIN.LS_Adv8 := FALSE;
   S708_TL_DC_PIN.LS_Ret8 := FALSE;
   S708_TL_DC_PIN.SOL_Adv := FALSE;
   S708_TL_DC_PIN.SOL_Ret := FALSE;
   S708_TL_DC_PIN.M_Ready := TRUE;
   S708_TL_DC_PIN.T_CHK1 := T#4S;
   S708_TL_DC_PIN.T_CHK2 := T#4S;
   S708_TL_DC_PIN.PB_Lamp_CHK := FALSE;
   S708_TL_DC_PIN.PB_Error_Rst := FALSE;
   S708_TL_DC_PIN.M_FLICK := FALSE;
   S708_TL_DC_PIN.M_Adv_Err := FALSE;
   S708_TL_DC_PIN.M_Ret_Err := FALSE;
   S708_TL_DC_PIN.LP_Adv := FALSE;
   S708_TL_DC_PIN.LP_Ret := FALSE;
   S708_TL_DC_PIN.Visu_Adv := W#16#0;
   S708_TL_DC_PIN.Visu_Ret := W#16#0;
   S708_TL_DC_PIN.Error_T1.IN := FALSE;
   S708_TL_DC_PIN.Error_T1.PT := T#4S;
   S708_TL_DC_PIN.Error_T1.Q := FALSE;
   S708_TL_DC_PIN.Error_T1.ET := T#0MS;
   S708_TL_DC_PIN.Error_T1.STATE := B#16#0;
   S708_TL_DC_PIN.Error_T1.STIME := T#23D5H8M48S439MS;
   S708_TL_DC_PIN.Error_T1.ATIME := T#23D5H8M48S920MS;
   S708_TL_DC_PIN.Error_T2.IN := FALSE;
   S708_TL_DC_PIN.Error_T2.PT := T#4S;
   S708_TL_DC_PIN.Error_T2.Q := FALSE;
   S708_TL_DC_PIN.Error_T2.ET := T#0MS;
   S708_TL_DC_PIN.Error_T2.STATE := B#16#0;
   S708_TL_DC_PIN.Error_T2.STIME := T#0MS;
   S708_TL_DC_PIN.Error_T2.ATIME := T#0MS;
   S708_TL_DC_PIN.Adv_End_Aux := FALSE;
   S708_TL_DC_PIN.Ret_End_Aux := FALSE;
   S708_TL_DC_PIN.CHK_Aux1 := FALSE;
   S708_TL_DC_PIN.CHK_Aux2 := FALSE;
   S708_TL_DC_PIN.Error_T1_DN := FALSE;
   S708_TL_DC_PIN.Error_T2_DN := FALSE;
   S708_TL_DC_PIN.Adv_Memo := FALSE;
   S708_TL_DC_PIN.Visu_Adv_Arr[0] := FALSE;
   S708_TL_DC_PIN.Visu_Adv_Arr[1] := FALSE;
   S708_TL_DC_PIN.Visu_Adv_Arr[2] := FALSE;
   S708_TL_DC_PIN.Visu_Adv_Arr[3] := FALSE;
   S708_TL_DC_PIN.Visu_Adv_Arr[4] := FALSE;
   S708_TL_DC_PIN.Visu_Adv_Arr[5] := FALSE;
   S708_TL_DC_PIN.Visu_Adv_Arr[6] := FALSE;
   S708_TL_DC_PIN.Visu_Adv_Arr[7] := FALSE;
   S708_TL_DC_PIN.Visu_Adv_Arr[8] := FALSE;
   S708_TL_DC_PIN.Visu_Adv_Arr[9] := FALSE;
   S708_TL_DC_PIN.Visu_Adv_Arr[10] := FALSE;
   S708_TL_DC_PIN.Visu_Adv_Arr[11] := FALSE;
   S708_TL_DC_PIN.Visu_Adv_Arr[12] := FALSE;
   S708_TL_DC_PIN.Visu_Adv_Arr[13] := FALSE;
   S708_TL_DC_PIN.Visu_Adv_Arr[14] := FALSE;
   S708_TL_DC_PIN.Visu_Adv_Arr[15] := FALSE;
   S708_TL_DC_PIN.Visu_Ret_Arr[0] := FALSE;
   S708_TL_DC_PIN.Visu_Ret_Arr[1] := FALSE;
   S708_TL_DC_PIN.Visu_Ret_Arr[2] := FALSE;
   S708_TL_DC_PIN.Visu_Ret_Arr[3] := FALSE;
   S708_TL_DC_PIN.Visu_Ret_Arr[4] := FALSE;
   S708_TL_DC_PIN.Visu_Ret_Arr[5] := FALSE;
   S708_TL_DC_PIN.Visu_Ret_Arr[6] := FALSE;
   S708_TL_DC_PIN.Visu_Ret_Arr[7] := FALSE;
   S708_TL_DC_PIN.Visu_Ret_Arr[8] := FALSE;
   S708_TL_DC_PIN.Visu_Ret_Arr[9] := FALSE;
   S708_TL_DC_PIN.Visu_Ret_Arr[10] := FALSE;
   S708_TL_DC_PIN.Visu_Ret_Arr[11] := FALSE;
   S708_TL_DC_PIN.Visu_Ret_Arr[12] := FALSE;
   S708_TL_DC_PIN.Visu_Ret_Arr[13] := FALSE;
   S708_TL_DC_PIN.Visu_Ret_Arr[14] := FALSE;
   S708_TL_DC_PIN.Visu_Ret_Arr[15] := FALSE;
   S708_TL_DC_PIN.BLK_Move_Ret := 0;
   S708_TL_DC_PIN.Enable := FALSE;
   S708_TL_DC_PIN.Adv_End := FALSE;
   S708_TL_DC_PIN.Ret_End := FALSE;
   S708_TL_DC_LATCH1.Enable_Aux := FALSE;
   S708_TL_DC_LATCH1.Adv_Amount := 5;
   S708_TL_DC_LATCH1.Ret_Amount := 5;
   S708_TL_DC_LATCH1.LS_Adv1 := FALSE;
   S708_TL_DC_LATCH1.LS_Ret1 := FALSE;
   S708_TL_DC_LATCH1.LS_Adv2 := FALSE;
   S708_TL_DC_LATCH1.LS_Ret2 := FALSE;
   S708_TL_DC_LATCH1.LS_Adv3 := FALSE;
   S708_TL_DC_LATCH1.LS_Ret3 := FALSE;
   S708_TL_DC_LATCH1.LS_Adv4 := FALSE;
   S708_TL_DC_LATCH1.LS_Ret4 := FALSE;
   S708_TL_DC_LATCH1.LS_Adv5 := FALSE;
   S708_TL_DC_LATCH1.LS_Ret5 := FALSE;
   S708_TL_DC_LATCH1.LS_Adv6 := FALSE;
   S708_TL_DC_LATCH1.LS_Ret6 := FALSE;
   S708_TL_DC_LATCH1.LS_Adv7 := FALSE;
   S708_TL_DC_LATCH1.LS_Ret7 := FALSE;
   S708_TL_DC_LATCH1.LS_Adv8 := FALSE;
   S708_TL_DC_LATCH1.LS_Ret8 := FALSE;
   S708_TL_DC_LATCH1.SOL_Adv := FALSE;
   S708_TL_DC_LATCH1.SOL_Ret := FALSE;
   S708_TL_DC_LATCH1.M_Ready := TRUE;
   S708_TL_DC_LATCH1.T_CHK1 := T#4S;
   S708_TL_DC_LATCH1.T_CHK2 := T#4S;
   S708_TL_DC_LATCH1.PB_Lamp_CHK := FALSE;
   S708_TL_DC_LATCH1.PB_Error_Rst := FALSE;
   S708_TL_DC_LATCH1.M_FLICK := FALSE;
   S708_TL_DC_LATCH1.M_Adv_Err := FALSE;
   S708_TL_DC_LATCH1.M_Ret_Err := FALSE;
   S708_TL_DC_LATCH1.LP_Adv := FALSE;
   S708_TL_DC_LATCH1.LP_Ret := FALSE;
   S708_TL_DC_LATCH1.Visu_Adv := W#16#0;
   S708_TL_DC_LATCH1.Visu_Ret := W#16#0;
   S708_TL_DC_LATCH1.Error_T1.IN := FALSE;
   S708_TL_DC_LATCH1.Error_T1.PT := T#4S;
   S708_TL_DC_LATCH1.Error_T1.Q := FALSE;
   S708_TL_DC_LATCH1.Error_T1.ET := T#0MS;
   S708_TL_DC_LATCH1.Error_T1.STATE := B#16#0;
   S708_TL_DC_LATCH1.Error_T1.STIME := T#23D5H8M50S20MS;
   S708_TL_DC_LATCH1.Error_T1.ATIME := T#23D5H8M51S531MS;
   S708_TL_DC_LATCH1.Error_T2.IN := FALSE;
   S708_TL_DC_LATCH1.Error_T2.PT := T#4S;
   S708_TL_DC_LATCH1.Error_T2.Q := FALSE;
   S708_TL_DC_LATCH1.Error_T2.ET := T#0MS;
   S708_TL_DC_LATCH1.Error_T2.STATE := B#16#0;
   S708_TL_DC_LATCH1.Error_T2.STIME := T#0MS;
   S708_TL_DC_LATCH1.Error_T2.ATIME := T#0MS;
   S708_TL_DC_LATCH1.Adv_End_Aux := FALSE;
   S708_TL_DC_LATCH1.Ret_End_Aux := FALSE;
   S708_TL_DC_LATCH1.CHK_Aux1 := FALSE;
   S708_TL_DC_LATCH1.CHK_Aux2 := FALSE;
   S708_TL_DC_LATCH1.Error_T1_DN := FALSE;
   S708_TL_DC_LATCH1.Error_T2_DN := FALSE;
   S708_TL_DC_LATCH1.Adv_Memo := FALSE;
   S708_TL_DC_LATCH1.Visu_Adv_Arr[0] := FALSE;
   S708_TL_DC_LATCH1.Visu_Adv_Arr[1] := FALSE;
   S708_TL_DC_LATCH1.Visu_Adv_Arr[2] := FALSE;
   S708_TL_DC_LATCH1.Visu_Adv_Arr[3] := FALSE;
   S708_TL_DC_LATCH1.Visu_Adv_Arr[4] := FALSE;
   S708_TL_DC_LATCH1.Visu_Adv_Arr[5] := FALSE;
   S708_TL_DC_LATCH1.Visu_Adv_Arr[6] := FALSE;
   S708_TL_DC_LATCH1.Visu_Adv_Arr[7] := FALSE;
   S708_TL_DC_LATCH1.Visu_Adv_Arr[8] := FALSE;
   S708_TL_DC_LATCH1.Visu_Adv_Arr[9] := FALSE;
   S708_TL_DC_LATCH1.Visu_Adv_Arr[10] := FALSE;
   S708_TL_DC_LATCH1.Visu_Adv_Arr[11] := FALSE;
   S708_TL_DC_LATCH1.Visu_Adv_Arr[12] := FALSE;
   S708_TL_DC_LATCH1.Visu_Adv_Arr[13] := FALSE;
   S708_TL_DC_LATCH1.Visu_Adv_Arr[14] := FALSE;
   S708_TL_DC_LATCH1.Visu_Adv_Arr[15] := FALSE;
   S708_TL_DC_LATCH1.Visu_Ret_Arr[0] := FALSE;
   S708_TL_DC_LATCH1.Visu_Ret_Arr[1] := FALSE;
   S708_TL_DC_LATCH1.Visu_Ret_Arr[2] := FALSE;
   S708_TL_DC_LATCH1.Visu_Ret_Arr[3] := FALSE;
   S708_TL_DC_LATCH1.Visu_Ret_Arr[4] := FALSE;
   S708_TL_DC_LATCH1.Visu_Ret_Arr[5] := FALSE;
   S708_TL_DC_LATCH1.Visu_Ret_Arr[6] := FALSE;
   S708_TL_DC_LATCH1.Visu_Ret_Arr[7] := FALSE;
   S708_TL_DC_LATCH1.Visu_Ret_Arr[8] := FALSE;
   S708_TL_DC_LATCH1.Visu_Ret_Arr[9] := FALSE;
   S708_TL_DC_LATCH1.Visu_Ret_Arr[10] := FALSE;
   S708_TL_DC_LATCH1.Visu_Ret_Arr[11] := FALSE;
   S708_TL_DC_LATCH1.Visu_Ret_Arr[12] := FALSE;
   S708_TL_DC_LATCH1.Visu_Ret_Arr[13] := FALSE;
   S708_TL_DC_LATCH1.Visu_Ret_Arr[14] := FALSE;
   S708_TL_DC_LATCH1.Visu_Ret_Arr[15] := FALSE;
   S708_TL_DC_LATCH1.BLK_Move_Ret := 0;
   S708_TL_DC_LATCH1.Enable := FALSE;
   S708_TL_DC_LATCH1.Adv_End := FALSE;
   S708_TL_DC_LATCH1.Ret_End := FALSE;
   S708_TL_DC_LATCH2.Enable_Aux := FALSE;
   S708_TL_DC_LATCH2.Adv_Amount := 2;
   S708_TL_DC_LATCH2.Ret_Amount := 2;
   S708_TL_DC_LATCH2.LS_Adv1 := FALSE;
   S708_TL_DC_LATCH2.LS_Ret1 := FALSE;
   S708_TL_DC_LATCH2.LS_Adv2 := FALSE;
   S708_TL_DC_LATCH2.LS_Ret2 := FALSE;
   S708_TL_DC_LATCH2.LS_Adv3 := FALSE;
   S708_TL_DC_LATCH2.LS_Ret3 := FALSE;
   S708_TL_DC_LATCH2.LS_Adv4 := FALSE;
   S708_TL_DC_LATCH2.LS_Ret4 := FALSE;
   S708_TL_DC_LATCH2.LS_Adv5 := FALSE;
   S708_TL_DC_LATCH2.LS_Ret5 := FALSE;
   S708_TL_DC_LATCH2.LS_Adv6 := FALSE;
   S708_TL_DC_LATCH2.LS_Ret6 := FALSE;
   S708_TL_DC_LATCH2.LS_Adv7 := FALSE;
   S708_TL_DC_LATCH2.LS_Ret7 := FALSE;
   S708_TL_DC_LATCH2.LS_Adv8 := FALSE;
   S708_TL_DC_LATCH2.LS_Ret8 := FALSE;
   S708_TL_DC_LATCH2.SOL_Adv := FALSE;
   S708_TL_DC_LATCH2.SOL_Ret := FALSE;
   S708_TL_DC_LATCH2.M_Ready := TRUE;
   S708_TL_DC_LATCH2.T_CHK1 := T#4S;
   S708_TL_DC_LATCH2.T_CHK2 := T#4S;
   S708_TL_DC_LATCH2.PB_Lamp_CHK := FALSE;
   S708_TL_DC_LATCH2.PB_Error_Rst := FALSE;
   S708_TL_DC_LATCH2.M_FLICK := FALSE;
   S708_TL_DC_LATCH2.M_Adv_Err := FALSE;
   S708_TL_DC_LATCH2.M_Ret_Err := FALSE;
   S708_TL_DC_LATCH2.LP_Adv := FALSE;
   S708_TL_DC_LATCH2.LP_Ret := FALSE;
   S708_TL_DC_LATCH2.Visu_Adv := W#16#0;
   S708_TL_DC_LATCH2.Visu_Ret := W#16#0;
   S708_TL_DC_LATCH2.Error_T1.IN := FALSE;
   S708_TL_DC_LATCH2.Error_T1.PT := T#4S;
   S708_TL_DC_LATCH2.Error_T1.Q := FALSE;
   S708_TL_DC_LATCH2.Error_T1.ET := T#0MS;
   S708_TL_DC_LATCH2.Error_T1.STATE := B#16#0;
   S708_TL_DC_LATCH2.Error_T1.STIME := T#23D5H8M50S20MS;
   S708_TL_DC_LATCH2.Error_T1.ATIME := T#23D5H8M50S937MS;
   S708_TL_DC_LATCH2.Error_T2.IN := FALSE;
   S708_TL_DC_LATCH2.Error_T2.PT := T#4S;
   S708_TL_DC_LATCH2.Error_T2.Q := FALSE;
   S708_TL_DC_LATCH2.Error_T2.ET := T#0MS;
   S708_TL_DC_LATCH2.Error_T2.STATE := B#16#0;
   S708_TL_DC_LATCH2.Error_T2.STIME := T#0MS;
   S708_TL_DC_LATCH2.Error_T2.ATIME := T#0MS;
   S708_TL_DC_LATCH2.Adv_End_Aux := FALSE;
   S708_TL_DC_LATCH2.Ret_End_Aux := FALSE;
   S708_TL_DC_LATCH2.CHK_Aux1 := FALSE;
   S708_TL_DC_LATCH2.CHK_Aux2 := FALSE;
   S708_TL_DC_LATCH2.Error_T1_DN := FALSE;
   S708_TL_DC_LATCH2.Error_T2_DN := FALSE;
   S708_TL_DC_LATCH2.Adv_Memo := FALSE;
   S708_TL_DC_LATCH2.Visu_Adv_Arr[0] := FALSE;
   S708_TL_DC_LATCH2.Visu_Adv_Arr[1] := FALSE;
   S708_TL_DC_LATCH2.Visu_Adv_Arr[2] := FALSE;
   S708_TL_DC_LATCH2.Visu_Adv_Arr[3] := FALSE;
   S708_TL_DC_LATCH2.Visu_Adv_Arr[4] := FALSE;
   S708_TL_DC_LATCH2.Visu_Adv_Arr[5] := FALSE;
   S708_TL_DC_LATCH2.Visu_Adv_Arr[6] := FALSE;
   S708_TL_DC_LATCH2.Visu_Adv_Arr[7] := FALSE;
   S708_TL_DC_LATCH2.Visu_Adv_Arr[8] := FALSE;
   S708_TL_DC_LATCH2.Visu_Adv_Arr[9] := FALSE;
   S708_TL_DC_LATCH2.Visu_Adv_Arr[10] := FALSE;
   S708_TL_DC_LATCH2.Visu_Adv_Arr[11] := FALSE;
   S708_TL_DC_LATCH2.Visu_Adv_Arr[12] := FALSE;
   S708_TL_DC_LATCH2.Visu_Adv_Arr[13] := FALSE;
   S708_TL_DC_LATCH2.Visu_Adv_Arr[14] := FALSE;
   S708_TL_DC_LATCH2.Visu_Adv_Arr[15] := FALSE;
   S708_TL_DC_LATCH2.Visu_Ret_Arr[0] := FALSE;
   S708_TL_DC_LATCH2.Visu_Ret_Arr[1] := FALSE;
   S708_TL_DC_LATCH2.Visu_Ret_Arr[2] := FALSE;
   S708_TL_DC_LATCH2.Visu_Ret_Arr[3] := FALSE;
   S708_TL_DC_LATCH2.Visu_Ret_Arr[4] := FALSE;
   S708_TL_DC_LATCH2.Visu_Ret_Arr[5] := FALSE;
   S708_TL_DC_LATCH2.Visu_Ret_Arr[6] := FALSE;
   S708_TL_DC_LATCH2.Visu_Ret_Arr[7] := FALSE;
   S708_TL_DC_LATCH2.Visu_Ret_Arr[8] := FALSE;
   S708_TL_DC_LATCH2.Visu_Ret_Arr[9] := FALSE;
   S708_TL_DC_LATCH2.Visu_Ret_Arr[10] := FALSE;
   S708_TL_DC_LATCH2.Visu_Ret_Arr[11] := FALSE;
   S708_TL_DC_LATCH2.Visu_Ret_Arr[12] := FALSE;
   S708_TL_DC_LATCH2.Visu_Ret_Arr[13] := FALSE;
   S708_TL_DC_LATCH2.Visu_Ret_Arr[14] := FALSE;
   S708_TL_DC_LATCH2.Visu_Ret_Arr[15] := FALSE;
   S708_TL_DC_LATCH2.BLK_Move_Ret := 0;
   S708_TL_DC_LATCH2.Enable := FALSE;
   S708_TL_DC_LATCH2.Adv_End := FALSE;
   S708_TL_DC_LATCH2.Ret_End := FALSE;
   S708_TL_DC_1ST_CLAMP1.Enable_Aux := FALSE;
   S708_TL_DC_1ST_CLAMP1.Adv_Amount := 1;
   S708_TL_DC_1ST_CLAMP1.Ret_Amount := 5;
   S708_TL_DC_1ST_CLAMP1.LS_Adv1 := FALSE;
   S708_TL_DC_1ST_CLAMP1.LS_Ret1 := FALSE;
   S708_TL_DC_1ST_CLAMP1.LS_Adv2 := FALSE;
   S708_TL_DC_1ST_CLAMP1.LS_Ret2 := FALSE;
   S708_TL_DC_1ST_CLAMP1.LS_Adv3 := FALSE;
   S708_TL_DC_1ST_CLAMP1.LS_Ret3 := FALSE;
   S708_TL_DC_1ST_CLAMP1.LS_Adv4 := FALSE;
   S708_TL_DC_1ST_CLAMP1.LS_Ret4 := FALSE;
   S708_TL_DC_1ST_CLAMP1.LS_Adv5 := FALSE;
   S708_TL_DC_1ST_CLAMP1.LS_Ret5 := FALSE;
   S708_TL_DC_1ST_CLAMP1.LS_Adv6 := FALSE;
   S708_TL_DC_1ST_CLAMP1.LS_Ret6 := FALSE;
   S708_TL_DC_1ST_CLAMP1.LS_Adv7 := FALSE;
   S708_TL_DC_1ST_CLAMP1.LS_Ret7 := FALSE;
   S708_TL_DC_1ST_CLAMP1.LS_Adv8 := FALSE;
   S708_TL_DC_1ST_CLAMP1.LS_Ret8 := FALSE;
   S708_TL_DC_1ST_CLAMP1.SOL_Adv := FALSE;
   S708_TL_DC_1ST_CLAMP1.SOL_Ret := FALSE;
   S708_TL_DC_1ST_CLAMP1.M_Ready := TRUE;
   S708_TL_DC_1ST_CLAMP1.T_CHK1 := T#4S;
   S708_TL_DC_1ST_CLAMP1.T_CHK2 := T#4S;
   S708_TL_DC_1ST_CLAMP1.PB_Lamp_CHK := FALSE;
   S708_TL_DC_1ST_CLAMP1.PB_Error_Rst := FALSE;
   S708_TL_DC_1ST_CLAMP1.M_FLICK := FALSE;
   S708_TL_DC_1ST_CLAMP1.M_Adv_Err := FALSE;
   S708_TL_DC_1ST_CLAMP1.M_Ret_Err := FALSE;
   S708_TL_DC_1ST_CLAMP1.LP_Adv := FALSE;
   S708_TL_DC_1ST_CLAMP1.LP_Ret := FALSE;
   S708_TL_DC_1ST_CLAMP1.Visu_Adv := W#16#0;
   S708_TL_DC_1ST_CLAMP1.Visu_Ret := W#16#0;
   S708_TL_DC_1ST_CLAMP1.Error_T1.IN := FALSE;
   S708_TL_DC_1ST_CLAMP1.Error_T1.PT := T#4S;
   S708_TL_DC_1ST_CLAMP1.Error_T1.Q := FALSE;
   S708_TL_DC_1ST_CLAMP1.Error_T1.ET := T#0MS;
   S708_TL_DC_1ST_CLAMP1.Error_T1.STATE := B#16#0;
   S708_TL_DC_1ST_CLAMP1.Error_T1.STIME := T#23D5H8M48S439MS;
   S708_TL_DC_1ST_CLAMP1.Error_T1.ATIME := T#23D5H8M49S975MS;
   S708_TL_DC_1ST_CLAMP1.Error_T2.IN := FALSE;
   S708_TL_DC_1ST_CLAMP1.Error_T2.PT := T#4S;
   S708_TL_DC_1ST_CLAMP1.Error_T2.Q := FALSE;
   S708_TL_DC_1ST_CLAMP1.Error_T2.ET := T#0MS;
   S708_TL_DC_1ST_CLAMP1.Error_T2.STATE := B#16#0;
   S708_TL_DC_1ST_CLAMP1.Error_T2.STIME := T#0MS;
   S708_TL_DC_1ST_CLAMP1.Error_T2.ATIME := T#0MS;
   S708_TL_DC_1ST_CLAMP1.Adv_End_Aux := FALSE;
   S708_TL_DC_1ST_CLAMP1.Ret_End_Aux := FALSE;
   S708_TL_DC_1ST_CLAMP1.CHK_Aux1 := FALSE;
   S708_TL_DC_1ST_CLAMP1.CHK_Aux2 := FALSE;
   S708_TL_DC_1ST_CLAMP1.Error_T1_DN := FALSE;
   S708_TL_DC_1ST_CLAMP1.Error_T2_DN := FALSE;
   S708_TL_DC_1ST_CLAMP1.Adv_Memo := FALSE;
   S708_TL_DC_1ST_CLAMP1.Visu_Adv_Arr[0] := FALSE;
   S708_TL_DC_1ST_CLAMP1.Visu_Adv_Arr[1] := FALSE;
   S708_TL_DC_1ST_CLAMP1.Visu_Adv_Arr[2] := FALSE;
   S708_TL_DC_1ST_CLAMP1.Visu_Adv_Arr[3] := FALSE;
   S708_TL_DC_1ST_CLAMP1.Visu_Adv_Arr[4] := FALSE;
   S708_TL_DC_1ST_CLAMP1.Visu_Adv_Arr[5] := FALSE;
   S708_TL_DC_1ST_CLAMP1.Visu_Adv_Arr[6] := FALSE;
   S708_TL_DC_1ST_CLAMP1.Visu_Adv_Arr[7] := FALSE;
   S708_TL_DC_1ST_CLAMP1.Visu_Adv_Arr[8] := FALSE;
   S708_TL_DC_1ST_CLAMP1.Visu_Adv_Arr[9] := FALSE;
   S708_TL_DC_1ST_CLAMP1.Visu_Adv_Arr[10] := FALSE;
   S708_TL_DC_1ST_CLAMP1.Visu_Adv_Arr[11] := FALSE;
   S708_TL_DC_1ST_CLAMP1.Visu_Adv_Arr[12] := FALSE;
   S708_TL_DC_1ST_CLAMP1.Visu_Adv_Arr[13] := FALSE;
   S708_TL_DC_1ST_CLAMP1.Visu_Adv_Arr[14] := FALSE;
   S708_TL_DC_1ST_CLAMP1.Visu_Adv_Arr[15] := FALSE;
   S708_TL_DC_1ST_CLAMP1.Visu_Ret_Arr[0] := FALSE;
   S708_TL_DC_1ST_CLAMP1.Visu_Ret_Arr[1] := FALSE;
   S708_TL_DC_1ST_CLAMP1.Visu_Ret_Arr[2] := FALSE;
   S708_TL_DC_1ST_CLAMP1.Visu_Ret_Arr[3] := FALSE;
   S708_TL_DC_1ST_CLAMP1.Visu_Ret_Arr[4] := FALSE;
   S708_TL_DC_1ST_CLAMP1.Visu_Ret_Arr[5] := FALSE;
   S708_TL_DC_1ST_CLAMP1.Visu_Ret_Arr[6] := FALSE;
   S708_TL_DC_1ST_CLAMP1.Visu_Ret_Arr[7] := FALSE;
   S708_TL_DC_1ST_CLAMP1.Visu_Ret_Arr[8] := FALSE;
   S708_TL_DC_1ST_CLAMP1.Visu_Ret_Arr[9] := FALSE;
   S708_TL_DC_1ST_CLAMP1.Visu_Ret_Arr[10] := FALSE;
   S708_TL_DC_1ST_CLAMP1.Visu_Ret_Arr[11] := FALSE;
   S708_TL_DC_1ST_CLAMP1.Visu_Ret_Arr[12] := FALSE;
   S708_TL_DC_1ST_CLAMP1.Visu_Ret_Arr[13] := FALSE;
   S708_TL_DC_1ST_CLAMP1.Visu_Ret_Arr[14] := FALSE;
   S708_TL_DC_1ST_CLAMP1.Visu_Ret_Arr[15] := FALSE;
   S708_TL_DC_1ST_CLAMP1.BLK_Move_Ret := 0;
   S708_TL_DC_1ST_CLAMP1.Enable := FALSE;
   S708_TL_DC_1ST_CLAMP1.Adv_End := FALSE;
   S708_TL_DC_1ST_CLAMP1.Ret_End := FALSE;
   S708_TL_DC_1ST_CLAMP2.Enable_Aux := FALSE;
   S708_TL_DC_1ST_CLAMP2.Adv_Amount := 1;
   S708_TL_DC_1ST_CLAMP2.Ret_Amount := 5;
   S708_TL_DC_1ST_CLAMP2.LS_Adv1 := FALSE;
   S708_TL_DC_1ST_CLAMP2.LS_Ret1 := FALSE;
   S708_TL_DC_1ST_CLAMP2.LS_Adv2 := FALSE;
   S708_TL_DC_1ST_CLAMP2.LS_Ret2 := FALSE;
   S708_TL_DC_1ST_CLAMP2.LS_Adv3 := FALSE;
   S708_TL_DC_1ST_CLAMP2.LS_Ret3 := FALSE;
   S708_TL_DC_1ST_CLAMP2.LS_Adv4 := FALSE;
   S708_TL_DC_1ST_CLAMP2.LS_Ret4 := FALSE;
   S708_TL_DC_1ST_CLAMP2.LS_Adv5 := FALSE;
   S708_TL_DC_1ST_CLAMP2.LS_Ret5 := FALSE;
   S708_TL_DC_1ST_CLAMP2.LS_Adv6 := FALSE;
   S708_TL_DC_1ST_CLAMP2.LS_Ret6 := FALSE;
   S708_TL_DC_1ST_CLAMP2.LS_Adv7 := FALSE;
   S708_TL_DC_1ST_CLAMP2.LS_Ret7 := FALSE;
   S708_TL_DC_1ST_CLAMP2.LS_Adv8 := FALSE;
   S708_TL_DC_1ST_CLAMP2.LS_Ret8 := FALSE;
   S708_TL_DC_1ST_CLAMP2.SOL_Adv := FALSE;
   S708_TL_DC_1ST_CLAMP2.SOL_Ret := FALSE;
   S708_TL_DC_1ST_CLAMP2.M_Ready := TRUE;
   S708_TL_DC_1ST_CLAMP2.T_CHK1 := T#4S;
   S708_TL_DC_1ST_CLAMP2.T_CHK2 := T#4S;
   S708_TL_DC_1ST_CLAMP2.PB_Lamp_CHK := FALSE;
   S708_TL_DC_1ST_CLAMP2.PB_Error_Rst := FALSE;
   S708_TL_DC_1ST_CLAMP2.M_FLICK := FALSE;
   S708_TL_DC_1ST_CLAMP2.M_Adv_Err := FALSE;
   S708_TL_DC_1ST_CLAMP2.M_Ret_Err := FALSE;
   S708_TL_DC_1ST_CLAMP2.LP_Adv := FALSE;
   S708_TL_DC_1ST_CLAMP2.LP_Ret := FALSE;
   S708_TL_DC_1ST_CLAMP2.Visu_Adv := W#16#0;
   S708_TL_DC_1ST_CLAMP2.Visu_Ret := W#16#0;
   S708_TL_DC_1ST_CLAMP2.Error_T1.IN := FALSE;
   S708_TL_DC_1ST_CLAMP2.Error_T1.PT := T#4S;
   S708_TL_DC_1ST_CLAMP2.Error_T1.Q := FALSE;
   S708_TL_DC_1ST_CLAMP2.Error_T1.ET := T#0MS;
   S708_TL_DC_1ST_CLAMP2.Error_T1.STATE := B#16#0;
   S708_TL_DC_1ST_CLAMP2.Error_T1.STIME := T#23D5H8M48S439MS;
   S708_TL_DC_1ST_CLAMP2.Error_T1.ATIME := T#23D5H8M49S699MS;
   S708_TL_DC_1ST_CLAMP2.Error_T2.IN := FALSE;
   S708_TL_DC_1ST_CLAMP2.Error_T2.PT := T#4S;
   S708_TL_DC_1ST_CLAMP2.Error_T2.Q := FALSE;
   S708_TL_DC_1ST_CLAMP2.Error_T2.ET := T#0MS;
   S708_TL_DC_1ST_CLAMP2.Error_T2.STATE := B#16#0;
   S708_TL_DC_1ST_CLAMP2.Error_T2.STIME := T#0MS;
   S708_TL_DC_1ST_CLAMP2.Error_T2.ATIME := T#0MS;
   S708_TL_DC_1ST_CLAMP2.Adv_End_Aux := FALSE;
   S708_TL_DC_1ST_CLAMP2.Ret_End_Aux := FALSE;
   S708_TL_DC_1ST_CLAMP2.CHK_Aux1 := FALSE;
   S708_TL_DC_1ST_CLAMP2.CHK_Aux2 := FALSE;
   S708_TL_DC_1ST_CLAMP2.Error_T1_DN := FALSE;
   S708_TL_DC_1ST_CLAMP2.Error_T2_DN := FALSE;
   S708_TL_DC_1ST_CLAMP2.Adv_Memo := FALSE;
   S708_TL_DC_1ST_CLAMP2.Visu_Adv_Arr[0] := FALSE;
   S708_TL_DC_1ST_CLAMP2.Visu_Adv_Arr[1] := FALSE;
   S708_TL_DC_1ST_CLAMP2.Visu_Adv_Arr[2] := FALSE;
   S708_TL_DC_1ST_CLAMP2.Visu_Adv_Arr[3] := FALSE;
   S708_TL_DC_1ST_CLAMP2.Visu_Adv_Arr[4] := FALSE;
   S708_TL_DC_1ST_CLAMP2.Visu_Adv_Arr[5] := FALSE;
   S708_TL_DC_1ST_CLAMP2.Visu_Adv_Arr[6] := FALSE;
   S708_TL_DC_1ST_CLAMP2.Visu_Adv_Arr[7] := FALSE;
   S708_TL_DC_1ST_CLAMP2.Visu_Adv_Arr[8] := FALSE;
   S708_TL_DC_1ST_CLAMP2.Visu_Adv_Arr[9] := FALSE;
   S708_TL_DC_1ST_CLAMP2.Visu_Adv_Arr[10] := FALSE;
   S708_TL_DC_1ST_CLAMP2.Visu_Adv_Arr[11] := FALSE;
   S708_TL_DC_1ST_CLAMP2.Visu_Adv_Arr[12] := FALSE;
   S708_TL_DC_1ST_CLAMP2.Visu_Adv_Arr[13] := FALSE;
   S708_TL_DC_1ST_CLAMP2.Visu_Adv_Arr[14] := FALSE;
   S708_TL_DC_1ST_CLAMP2.Visu_Adv_Arr[15] := FALSE;
   S708_TL_DC_1ST_CLAMP2.Visu_Ret_Arr[0] := FALSE;
   S708_TL_DC_1ST_CLAMP2.Visu_Ret_Arr[1] := FALSE;
   S708_TL_DC_1ST_CLAMP2.Visu_Ret_Arr[2] := FALSE;
   S708_TL_DC_1ST_CLAMP2.Visu_Ret_Arr[3] := FALSE;
   S708_TL_DC_1ST_CLAMP2.Visu_Ret_Arr[4] := FALSE;
   S708_TL_DC_1ST_CLAMP2.Visu_Ret_Arr[5] := FALSE;
   S708_TL_DC_1ST_CLAMP2.Visu_Ret_Arr[6] := FALSE;
   S708_TL_DC_1ST_CLAMP2.Visu_Ret_Arr[7] := FALSE;
   S708_TL_DC_1ST_CLAMP2.Visu_Ret_Arr[8] := FALSE;
   S708_TL_DC_1ST_CLAMP2.Visu_Ret_Arr[9] := FALSE;
   S708_TL_DC_1ST_CLAMP2.Visu_Ret_Arr[10] := FALSE;
   S708_TL_DC_1ST_CLAMP2.Visu_Ret_Arr[11] := FALSE;
   S708_TL_DC_1ST_CLAMP2.Visu_Ret_Arr[12] := FALSE;
   S708_TL_DC_1ST_CLAMP2.Visu_Ret_Arr[13] := FALSE;
   S708_TL_DC_1ST_CLAMP2.Visu_Ret_Arr[14] := FALSE;
   S708_TL_DC_1ST_CLAMP2.Visu_Ret_Arr[15] := FALSE;
   S708_TL_DC_1ST_CLAMP2.BLK_Move_Ret := 0;
   S708_TL_DC_1ST_CLAMP2.Enable := FALSE;
   S708_TL_DC_1ST_CLAMP2.Adv_End := FALSE;
   S708_TL_DC_1ST_CLAMP2.Ret_End := FALSE;
   S708_TL_DC_1ST_CLAMP3.Enable_Aux := FALSE;
   S708_TL_DC_1ST_CLAMP3.Adv_Amount := 1;
   S708_TL_DC_1ST_CLAMP3.Ret_Amount := 3;
   S708_TL_DC_1ST_CLAMP3.LS_Adv1 := FALSE;
   S708_TL_DC_1ST_CLAMP3.LS_Ret1 := FALSE;
   S708_TL_DC_1ST_CLAMP3.LS_Adv2 := FALSE;
   S708_TL_DC_1ST_CLAMP3.LS_Ret2 := FALSE;
   S708_TL_DC_1ST_CLAMP3.LS_Adv3 := FALSE;
   S708_TL_DC_1ST_CLAMP3.LS_Ret3 := FALSE;
   S708_TL_DC_1ST_CLAMP3.LS_Adv4 := FALSE;
   S708_TL_DC_1ST_CLAMP3.LS_Ret4 := FALSE;
   S708_TL_DC_1ST_CLAMP3.LS_Adv5 := FALSE;
   S708_TL_DC_1ST_CLAMP3.LS_Ret5 := FALSE;
   S708_TL_DC_1ST_CLAMP3.LS_Adv6 := FALSE;
   S708_TL_DC_1ST_CLAMP3.LS_Ret6 := FALSE;
   S708_TL_DC_1ST_CLAMP3.LS_Adv7 := FALSE;
   S708_TL_DC_1ST_CLAMP3.LS_Ret7 := FALSE;
   S708_TL_DC_1ST_CLAMP3.LS_Adv8 := FALSE;
   S708_TL_DC_1ST_CLAMP3.LS_Ret8 := FALSE;
   S708_TL_DC_1ST_CLAMP3.SOL_Adv := FALSE;
   S708_TL_DC_1ST_CLAMP3.SOL_Ret := FALSE;
   S708_TL_DC_1ST_CLAMP3.M_Ready := TRUE;
   S708_TL_DC_1ST_CLAMP3.T_CHK1 := T#4S;
   S708_TL_DC_1ST_CLAMP3.T_CHK2 := T#4S;
   S708_TL_DC_1ST_CLAMP3.PB_Lamp_CHK := FALSE;
   S708_TL_DC_1ST_CLAMP3.PB_Error_Rst := FALSE;
   S708_TL_DC_1ST_CLAMP3.M_FLICK := FALSE;
   S708_TL_DC_1ST_CLAMP3.M_Adv_Err := FALSE;
   S708_TL_DC_1ST_CLAMP3.M_Ret_Err := FALSE;
   S708_TL_DC_1ST_CLAMP3.LP_Adv := FALSE;
   S708_TL_DC_1ST_CLAMP3.LP_Ret := FALSE;
   S708_TL_DC_1ST_CLAMP3.Visu_Adv := W#16#0;
   S708_TL_DC_1ST_CLAMP3.Visu_Ret := W#16#0;
   S708_TL_DC_1ST_CLAMP3.Error_T1.IN := FALSE;
   S708_TL_DC_1ST_CLAMP3.Error_T1.PT := T#4S;
   S708_TL_DC_1ST_CLAMP3.Error_T1.Q := FALSE;
   S708_TL_DC_1ST_CLAMP3.Error_T1.ET := T#0MS;
   S708_TL_DC_1ST_CLAMP3.Error_T1.STATE := B#16#0;
   S708_TL_DC_1ST_CLAMP3.Error_T1.STIME := T#23D5H8M48S439MS;
   S708_TL_DC_1ST_CLAMP3.Error_T1.ATIME := T#23D5H8M49S975MS;
   S708_TL_DC_1ST_CLAMP3.Error_T2.IN := FALSE;
   S708_TL_DC_1ST_CLAMP3.Error_T2.PT := T#4S;
   S708_TL_DC_1ST_CLAMP3.Error_T2.Q := FALSE;
   S708_TL_DC_1ST_CLAMP3.Error_T2.ET := T#0MS;
   S708_TL_DC_1ST_CLAMP3.Error_T2.STATE := B#16#0;
   S708_TL_DC_1ST_CLAMP3.Error_T2.STIME := T#0MS;
   S708_TL_DC_1ST_CLAMP3.Error_T2.ATIME := T#0MS;
   S708_TL_DC_1ST_CLAMP3.Adv_End_Aux := FALSE;
   S708_TL_DC_1ST_CLAMP3.Ret_End_Aux := FALSE;
   S708_TL_DC_1ST_CLAMP3.CHK_Aux1 := FALSE;
   S708_TL_DC_1ST_CLAMP3.CHK_Aux2 := FALSE;
   S708_TL_DC_1ST_CLAMP3.Error_T1_DN := FALSE;
   S708_TL_DC_1ST_CLAMP3.Error_T2_DN := FALSE;
   S708_TL_DC_1ST_CLAMP3.Adv_Memo := FALSE;
   S708_TL_DC_1ST_CLAMP3.Visu_Adv_Arr[0] := FALSE;
   S708_TL_DC_1ST_CLAMP3.Visu_Adv_Arr[1] := FALSE;
   S708_TL_DC_1ST_CLAMP3.Visu_Adv_Arr[2] := FALSE;
   S708_TL_DC_1ST_CLAMP3.Visu_Adv_Arr[3] := FALSE;
   S708_TL_DC_1ST_CLAMP3.Visu_Adv_Arr[4] := FALSE;
   S708_TL_DC_1ST_CLAMP3.Visu_Adv_Arr[5] := FALSE;
   S708_TL_DC_1ST_CLAMP3.Visu_Adv_Arr[6] := FALSE;
   S708_TL_DC_1ST_CLAMP3.Visu_Adv_Arr[7] := FALSE;
   S708_TL_DC_1ST_CLAMP3.Visu_Adv_Arr[8] := FALSE;
   S708_TL_DC_1ST_CLAMP3.Visu_Adv_Arr[9] := FALSE;
   S708_TL_DC_1ST_CLAMP3.Visu_Adv_Arr[10] := FALSE;
   S708_TL_DC_1ST_CLAMP3.Visu_Adv_Arr[11] := FALSE;
   S708_TL_DC_1ST_CLAMP3.Visu_Adv_Arr[12] := FALSE;
   S708_TL_DC_1ST_CLAMP3.Visu_Adv_Arr[13] := FALSE;
   S708_TL_DC_1ST_CLAMP3.Visu_Adv_Arr[14] := FALSE;
   S708_TL_DC_1ST_CLAMP3.Visu_Adv_Arr[15] := FALSE;
   S708_TL_DC_1ST_CLAMP3.Visu_Ret_Arr[0] := FALSE;
   S708_TL_DC_1ST_CLAMP3.Visu_Ret_Arr[1] := FALSE;
   S708_TL_DC_1ST_CLAMP3.Visu_Ret_Arr[2] := FALSE;
   S708_TL_DC_1ST_CLAMP3.Visu_Ret_Arr[3] := FALSE;
   S708_TL_DC_1ST_CLAMP3.Visu_Ret_Arr[4] := FALSE;
   S708_TL_DC_1ST_CLAMP3.Visu_Ret_Arr[5] := FALSE;
   S708_TL_DC_1ST_CLAMP3.Visu_Ret_Arr[6] := FALSE;
   S708_TL_DC_1ST_CLAMP3.Visu_Ret_Arr[7] := FALSE;
   S708_TL_DC_1ST_CLAMP3.Visu_Ret_Arr[8] := FALSE;
   S708_TL_DC_1ST_CLAMP3.Visu_Ret_Arr[9] := FALSE;
   S708_TL_DC_1ST_CLAMP3.Visu_Ret_Arr[10] := FALSE;
   S708_TL_DC_1ST_CLAMP3.Visu_Ret_Arr[11] := FALSE;
   S708_TL_DC_1ST_CLAMP3.Visu_Ret_Arr[12] := FALSE;
   S708_TL_DC_1ST_CLAMP3.Visu_Ret_Arr[13] := FALSE;
   S708_TL_DC_1ST_CLAMP3.Visu_Ret_Arr[14] := FALSE;
   S708_TL_DC_1ST_CLAMP3.Visu_Ret_Arr[15] := FALSE;
   S708_TL_DC_1ST_CLAMP3.BLK_Move_Ret := 0;
   S708_TL_DC_1ST_CLAMP3.Enable := FALSE;
   S708_TL_DC_1ST_CLAMP3.Adv_End := FALSE;
   S708_TL_DC_1ST_CLAMP3.Ret_End := FALSE;
   S708_TL_DC_2ND_CLAMP1.Enable_Aux := FALSE;
   S708_TL_DC_2ND_CLAMP1.Adv_Amount := 1;
   S708_TL_DC_2ND_CLAMP1.Ret_Amount := 5;
   S708_TL_DC_2ND_CLAMP1.LS_Adv1 := FALSE;
   S708_TL_DC_2ND_CLAMP1.LS_Ret1 := FALSE;
   S708_TL_DC_2ND_CLAMP1.LS_Adv2 := FALSE;
   S708_TL_DC_2ND_CLAMP1.LS_Ret2 := FALSE;
   S708_TL_DC_2ND_CLAMP1.LS_Adv3 := FALSE;
   S708_TL_DC_2ND_CLAMP1.LS_Ret3 := FALSE;
   S708_TL_DC_2ND_CLAMP1.LS_Adv4 := FALSE;
   S708_TL_DC_2ND_CLAMP1.LS_Ret4 := FALSE;
   S708_TL_DC_2ND_CLAMP1.LS_Adv5 := FALSE;
   S708_TL_DC_2ND_CLAMP1.LS_Ret5 := FALSE;
   S708_TL_DC_2ND_CLAMP1.LS_Adv6 := FALSE;
   S708_TL_DC_2ND_CLAMP1.LS_Ret6 := FALSE;
   S708_TL_DC_2ND_CLAMP1.LS_Adv7 := FALSE;
   S708_TL_DC_2ND_CLAMP1.LS_Ret7 := FALSE;
   S708_TL_DC_2ND_CLAMP1.LS_Adv8 := FALSE;
   S708_TL_DC_2ND_CLAMP1.LS_Ret8 := FALSE;
   S708_TL_DC_2ND_CLAMP1.SOL_Adv := FALSE;
   S708_TL_DC_2ND_CLAMP1.SOL_Ret := FALSE;
   S708_TL_DC_2ND_CLAMP1.M_Ready := TRUE;
   S708_TL_DC_2ND_CLAMP1.T_CHK1 := T#4S;
   S708_TL_DC_2ND_CLAMP1.T_CHK2 := T#4S;
   S708_TL_DC_2ND_CLAMP1.PB_Lamp_CHK := FALSE;
   S708_TL_DC_2ND_CLAMP1.PB_Error_Rst := FALSE;
   S708_TL_DC_2ND_CLAMP1.M_FLICK := FALSE;
   S708_TL_DC_2ND_CLAMP1.M_Adv_Err := FALSE;
   S708_TL_DC_2ND_CLAMP1.M_Ret_Err := FALSE;
   S708_TL_DC_2ND_CLAMP1.LP_Adv := FALSE;
   S708_TL_DC_2ND_CLAMP1.LP_Ret := FALSE;
   S708_TL_DC_2ND_CLAMP1.Visu_Adv := W#16#0;
   S708_TL_DC_2ND_CLAMP1.Visu_Ret := W#16#0;
   S708_TL_DC_2ND_CLAMP1.Error_T1.IN := FALSE;
   S708_TL_DC_2ND_CLAMP1.Error_T1.PT := T#4S;
   S708_TL_DC_2ND_CLAMP1.Error_T1.Q := FALSE;
   S708_TL_DC_2ND_CLAMP1.Error_T1.ET := T#0MS;
   S708_TL_DC_2ND_CLAMP1.Error_T1.STATE := B#16#0;
   S708_TL_DC_2ND_CLAMP1.Error_T1.STIME := T#23D5H8M48S439MS;
   S708_TL_DC_2ND_CLAMP1.Error_T1.ATIME := T#23D5H8M49S792MS;
   S708_TL_DC_2ND_CLAMP1.Error_T2.IN := FALSE;
   S708_TL_DC_2ND_CLAMP1.Error_T2.PT := T#4S;
   S708_TL_DC_2ND_CLAMP1.Error_T2.Q := FALSE;
   S708_TL_DC_2ND_CLAMP1.Error_T2.ET := T#0MS;
   S708_TL_DC_2ND_CLAMP1.Error_T2.STATE := B#16#0;
   S708_TL_DC_2ND_CLAMP1.Error_T2.STIME := T#0MS;
   S708_TL_DC_2ND_CLAMP1.Error_T2.ATIME := T#0MS;
   S708_TL_DC_2ND_CLAMP1.Adv_End_Aux := FALSE;
   S708_TL_DC_2ND_CLAMP1.Ret_End_Aux := FALSE;
   S708_TL_DC_2ND_CLAMP1.CHK_Aux1 := FALSE;
   S708_TL_DC_2ND_CLAMP1.CHK_Aux2 := FALSE;
   S708_TL_DC_2ND_CLAMP1.Error_T1_DN := FALSE;
   S708_TL_DC_2ND_CLAMP1.Error_T2_DN := FALSE;
   S708_TL_DC_2ND_CLAMP1.Adv_Memo := FALSE;
   S708_TL_DC_2ND_CLAMP1.Visu_Adv_Arr[0] := FALSE;
   S708_TL_DC_2ND_CLAMP1.Visu_Adv_Arr[1] := FALSE;
   S708_TL_DC_2ND_CLAMP1.Visu_Adv_Arr[2] := FALSE;
   S708_TL_DC_2ND_CLAMP1.Visu_Adv_Arr[3] := FALSE;
   S708_TL_DC_2ND_CLAMP1.Visu_Adv_Arr[4] := FALSE;
   S708_TL_DC_2ND_CLAMP1.Visu_Adv_Arr[5] := FALSE;
   S708_TL_DC_2ND_CLAMP1.Visu_Adv_Arr[6] := FALSE;
   S708_TL_DC_2ND_CLAMP1.Visu_Adv_Arr[7] := FALSE;
   S708_TL_DC_2ND_CLAMP1.Visu_Adv_Arr[8] := FALSE;
   S708_TL_DC_2ND_CLAMP1.Visu_Adv_Arr[9] := FALSE;
   S708_TL_DC_2ND_CLAMP1.Visu_Adv_Arr[10] := FALSE;
   S708_TL_DC_2ND_CLAMP1.Visu_Adv_Arr[11] := FALSE;
   S708_TL_DC_2ND_CLAMP1.Visu_Adv_Arr[12] := FALSE;
   S708_TL_DC_2ND_CLAMP1.Visu_Adv_Arr[13] := FALSE;
   S708_TL_DC_2ND_CLAMP1.Visu_Adv_Arr[14] := FALSE;
   S708_TL_DC_2ND_CLAMP1.Visu_Adv_Arr[15] := FALSE;
   S708_TL_DC_2ND_CLAMP1.Visu_Ret_Arr[0] := FALSE;
   S708_TL_DC_2ND_CLAMP1.Visu_Ret_Arr[1] := FALSE;
   S708_TL_DC_2ND_CLAMP1.Visu_Ret_Arr[2] := FALSE;
   S708_TL_DC_2ND_CLAMP1.Visu_Ret_Arr[3] := FALSE;
   S708_TL_DC_2ND_CLAMP1.Visu_Ret_Arr[4] := FALSE;
   S708_TL_DC_2ND_CLAMP1.Visu_Ret_Arr[5] := FALSE;
   S708_TL_DC_2ND_CLAMP1.Visu_Ret_Arr[6] := FALSE;
   S708_TL_DC_2ND_CLAMP1.Visu_Ret_Arr[7] := FALSE;
   S708_TL_DC_2ND_CLAMP1.Visu_Ret_Arr[8] := FALSE;
   S708_TL_DC_2ND_CLAMP1.Visu_Ret_Arr[9] := FALSE;
   S708_TL_DC_2ND_CLAMP1.Visu_Ret_Arr[10] := FALSE;
   S708_TL_DC_2ND_CLAMP1.Visu_Ret_Arr[11] := FALSE;
   S708_TL_DC_2ND_CLAMP1.Visu_Ret_Arr[12] := FALSE;
   S708_TL_DC_2ND_CLAMP1.Visu_Ret_Arr[13] := FALSE;
   S708_TL_DC_2ND_CLAMP1.Visu_Ret_Arr[14] := FALSE;
   S708_TL_DC_2ND_CLAMP1.Visu_Ret_Arr[15] := FALSE;
   S708_TL_DC_2ND_CLAMP1.BLK_Move_Ret := 0;
   S708_TL_DC_2ND_CLAMP1.Enable := FALSE;
   S708_TL_DC_2ND_CLAMP1.Adv_End := FALSE;
   S708_TL_DC_2ND_CLAMP1.Ret_End := FALSE;
   S708_TL_DC_2ND_CLAMP2.Enable_Aux := FALSE;
   S708_TL_DC_2ND_CLAMP2.Adv_Amount := 1;
   S708_TL_DC_2ND_CLAMP2.Ret_Amount := 5;
   S708_TL_DC_2ND_CLAMP2.LS_Adv1 := FALSE;
   S708_TL_DC_2ND_CLAMP2.LS_Ret1 := FALSE;
   S708_TL_DC_2ND_CLAMP2.LS_Adv2 := FALSE;
   S708_TL_DC_2ND_CLAMP2.LS_Ret2 := FALSE;
   S708_TL_DC_2ND_CLAMP2.LS_Adv3 := FALSE;
   S708_TL_DC_2ND_CLAMP2.LS_Ret3 := FALSE;
   S708_TL_DC_2ND_CLAMP2.LS_Adv4 := FALSE;
   S708_TL_DC_2ND_CLAMP2.LS_Ret4 := FALSE;
   S708_TL_DC_2ND_CLAMP2.LS_Adv5 := FALSE;
   S708_TL_DC_2ND_CLAMP2.LS_Ret5 := FALSE;
   S708_TL_DC_2ND_CLAMP2.LS_Adv6 := FALSE;
   S708_TL_DC_2ND_CLAMP2.LS_Ret6 := FALSE;
   S708_TL_DC_2ND_CLAMP2.LS_Adv7 := FALSE;
   S708_TL_DC_2ND_CLAMP2.LS_Ret7 := FALSE;
   S708_TL_DC_2ND_CLAMP2.LS_Adv8 := FALSE;
   S708_TL_DC_2ND_CLAMP2.LS_Ret8 := FALSE;
   S708_TL_DC_2ND_CLAMP2.SOL_Adv := FALSE;
   S708_TL_DC_2ND_CLAMP2.SOL_Ret := FALSE;
   S708_TL_DC_2ND_CLAMP2.M_Ready := TRUE;
   S708_TL_DC_2ND_CLAMP2.T_CHK1 := T#4S;
   S708_TL_DC_2ND_CLAMP2.T_CHK2 := T#4S;
   S708_TL_DC_2ND_CLAMP2.PB_Lamp_CHK := FALSE;
   S708_TL_DC_2ND_CLAMP2.PB_Error_Rst := FALSE;
   S708_TL_DC_2ND_CLAMP2.M_FLICK := FALSE;
   S708_TL_DC_2ND_CLAMP2.M_Adv_Err := FALSE;
   S708_TL_DC_2ND_CLAMP2.M_Ret_Err := FALSE;
   S708_TL_DC_2ND_CLAMP2.LP_Adv := FALSE;
   S708_TL_DC_2ND_CLAMP2.LP_Ret := FALSE;
   S708_TL_DC_2ND_CLAMP2.Visu_Adv := W#16#0;
   S708_TL_DC_2ND_CLAMP2.Visu_Ret := W#16#0;
   S708_TL_DC_2ND_CLAMP2.Error_T1.IN := FALSE;
   S708_TL_DC_2ND_CLAMP2.Error_T1.PT := T#4S;
   S708_TL_DC_2ND_CLAMP2.Error_T1.Q := FALSE;
   S708_TL_DC_2ND_CLAMP2.Error_T1.ET := T#0MS;
   S708_TL_DC_2ND_CLAMP2.Error_T1.STATE := B#16#0;
   S708_TL_DC_2ND_CLAMP2.Error_T1.STIME := T#23D5H8M48S439MS;
   S708_TL_DC_2ND_CLAMP2.Error_T1.ATIME := T#23D5H8M50S20MS;
   S708_TL_DC_2ND_CLAMP2.Error_T2.IN := FALSE;
   S708_TL_DC_2ND_CLAMP2.Error_T2.PT := T#4S;
   S708_TL_DC_2ND_CLAMP2.Error_T2.Q := FALSE;
   S708_TL_DC_2ND_CLAMP2.Error_T2.ET := T#0MS;
   S708_TL_DC_2ND_CLAMP2.Error_T2.STATE := B#16#0;
   S708_TL_DC_2ND_CLAMP2.Error_T2.STIME := T#0MS;
   S708_TL_DC_2ND_CLAMP2.Error_T2.ATIME := T#0MS;
   S708_TL_DC_2ND_CLAMP2.Adv_End_Aux := FALSE;
   S708_TL_DC_2ND_CLAMP2.Ret_End_Aux := FALSE;
   S708_TL_DC_2ND_CLAMP2.CHK_Aux1 := FALSE;
   S708_TL_DC_2ND_CLAMP2.CHK_Aux2 := FALSE;
   S708_TL_DC_2ND_CLAMP2.Error_T1_DN := FALSE;
   S708_TL_DC_2ND_CLAMP2.Error_T2_DN := FALSE;
   S708_TL_DC_2ND_CLAMP2.Adv_Memo := FALSE;
   S708_TL_DC_2ND_CLAMP2.Visu_Adv_Arr[0] := FALSE;
   S708_TL_DC_2ND_CLAMP2.Visu_Adv_Arr[1] := FALSE;
   S708_TL_DC_2ND_CLAMP2.Visu_Adv_Arr[2] := FALSE;
   S708_TL_DC_2ND_CLAMP2.Visu_Adv_Arr[3] := FALSE;
   S708_TL_DC_2ND_CLAMP2.Visu_Adv_Arr[4] := FALSE;
   S708_TL_DC_2ND_CLAMP2.Visu_Adv_Arr[5] := FALSE;
   S708_TL_DC_2ND_CLAMP2.Visu_Adv_Arr[6] := FALSE;
   S708_TL_DC_2ND_CLAMP2.Visu_Adv_Arr[7] := FALSE;
   S708_TL_DC_2ND_CLAMP2.Visu_Adv_Arr[8] := FALSE;
   S708_TL_DC_2ND_CLAMP2.Visu_Adv_Arr[9] := FALSE;
   S708_TL_DC_2ND_CLAMP2.Visu_Adv_Arr[10] := FALSE;
   S708_TL_DC_2ND_CLAMP2.Visu_Adv_Arr[11] := FALSE;
   S708_TL_DC_2ND_CLAMP2.Visu_Adv_Arr[12] := FALSE;
   S708_TL_DC_2ND_CLAMP2.Visu_Adv_Arr[13] := FALSE;
   S708_TL_DC_2ND_CLAMP2.Visu_Adv_Arr[14] := FALSE;
   S708_TL_DC_2ND_CLAMP2.Visu_Adv_Arr[15] := FALSE;
   S708_TL_DC_2ND_CLAMP2.Visu_Ret_Arr[0] := FALSE;
   S708_TL_DC_2ND_CLAMP2.Visu_Ret_Arr[1] := FALSE;
   S708_TL_DC_2ND_CLAMP2.Visu_Ret_Arr[2] := FALSE;
   S708_TL_DC_2ND_CLAMP2.Visu_Ret_Arr[3] := FALSE;
   S708_TL_DC_2ND_CLAMP2.Visu_Ret_Arr[4] := FALSE;
   S708_TL_DC_2ND_CLAMP2.Visu_Ret_Arr[5] := FALSE;
   S708_TL_DC_2ND_CLAMP2.Visu_Ret_Arr[6] := FALSE;
   S708_TL_DC_2ND_CLAMP2.Visu_Ret_Arr[7] := FALSE;
   S708_TL_DC_2ND_CLAMP2.Visu_Ret_Arr[8] := FALSE;
   S708_TL_DC_2ND_CLAMP2.Visu_Ret_Arr[9] := FALSE;
   S708_TL_DC_2ND_CLAMP2.Visu_Ret_Arr[10] := FALSE;
   S708_TL_DC_2ND_CLAMP2.Visu_Ret_Arr[11] := FALSE;
   S708_TL_DC_2ND_CLAMP2.Visu_Ret_Arr[12] := FALSE;
   S708_TL_DC_2ND_CLAMP2.Visu_Ret_Arr[13] := FALSE;
   S708_TL_DC_2ND_CLAMP2.Visu_Ret_Arr[14] := FALSE;
   S708_TL_DC_2ND_CLAMP2.Visu_Ret_Arr[15] := FALSE;
   S708_TL_DC_2ND_CLAMP2.BLK_Move_Ret := 0;
   S708_TL_DC_2ND_CLAMP2.Enable := FALSE;
   S708_TL_DC_2ND_CLAMP2.Adv_End := FALSE;
   S708_TL_DC_2ND_CLAMP2.Ret_End := FALSE;
   S708_TL_DC_U261.Enable_Aux := FALSE;
   S708_TL_DC_U261.Adv_Amount := 1;
   S708_TL_DC_U261.Ret_Amount := 1;
   S708_TL_DC_U261.LS_Adv1 := FALSE;
   S708_TL_DC_U261.LS_Ret1 := FALSE;
   S708_TL_DC_U261.LS_Adv2 := FALSE;
   S708_TL_DC_U261.LS_Ret2 := FALSE;
   S708_TL_DC_U261.LS_Adv3 := FALSE;
   S708_TL_DC_U261.LS_Ret3 := FALSE;
   S708_TL_DC_U261.LS_Adv4 := FALSE;
   S708_TL_DC_U261.LS_Ret4 := FALSE;
   S708_TL_DC_U261.LS_Adv5 := FALSE;
   S708_TL_DC_U261.LS_Ret5 := FALSE;
   S708_TL_DC_U261.LS_Adv6 := FALSE;
   S708_TL_DC_U261.LS_Ret6 := FALSE;
   S708_TL_DC_U261.LS_Adv7 := FALSE;
   S708_TL_DC_U261.LS_Ret7 := FALSE;
   S708_TL_DC_U261.LS_Adv8 := FALSE;
   S708_TL_DC_U261.LS_Ret8 := FALSE;
   S708_TL_DC_U261.SOL_Adv := FALSE;
   S708_TL_DC_U261.SOL_Ret := FALSE;
   S708_TL_DC_U261.M_Ready := TRUE;
   S708_TL_DC_U261.T_CHK1 := T#4S;
   S708_TL_DC_U261.T_CHK2 := T#4S;
   S708_TL_DC_U261.PB_Lamp_CHK := FALSE;
   S708_TL_DC_U261.PB_Error_Rst := FALSE;
   S708_TL_DC_U261.M_FLICK := TRUE;
   S708_TL_DC_U261.M_Adv_Err := FALSE;
   S708_TL_DC_U261.M_Ret_Err := FALSE;
   S708_TL_DC_U261.LP_Adv := FALSE;
   S708_TL_DC_U261.LP_Ret := FALSE;
   S708_TL_DC_U261.Visu_Adv := W#16#0;
   S708_TL_DC_U261.Visu_Ret := W#16#0;
   S708_TL_DC_U261.Error_T1.IN := FALSE;
   S708_TL_DC_U261.Error_T1.PT := T#4S;
   S708_TL_DC_U261.Error_T1.Q := FALSE;
   S708_TL_DC_U261.Error_T1.ET := T#0MS;
   S708_TL_DC_U261.Error_T1.STATE := B#16#0;
   S708_TL_DC_U261.Error_T1.STIME := T#23D5H8M49S747MS;
   S708_TL_DC_U261.Error_T1.ATIME := T#23D5H8M51S441MS;
   S708_TL_DC_U261.Error_T2.IN := FALSE;
   S708_TL_DC_U261.Error_T2.PT := T#4S;
   S708_TL_DC_U261.Error_T2.Q := FALSE;
   S708_TL_DC_U261.Error_T2.ET := T#0MS;
   S708_TL_DC_U261.Error_T2.STATE := B#16#0;
   S708_TL_DC_U261.Error_T2.STIME := T#0MS;
   S708_TL_DC_U261.Error_T2.ATIME := T#0MS;
   S708_TL_DC_U261.Adv_End_Aux := FALSE;
   S708_TL_DC_U261.Ret_End_Aux := FALSE;
   S708_TL_DC_U261.CHK_Aux1 := FALSE;
   S708_TL_DC_U261.CHK_Aux2 := FALSE;
   S708_TL_DC_U261.Error_T1_DN := FALSE;
   S708_TL_DC_U261.Error_T2_DN := FALSE;
   S708_TL_DC_U261.Adv_Memo := FALSE;
   S708_TL_DC_U261.Visu_Adv_Arr[0] := FALSE;
   S708_TL_DC_U261.Visu_Adv_Arr[1] := FALSE;
   S708_TL_DC_U261.Visu_Adv_Arr[2] := FALSE;
   S708_TL_DC_U261.Visu_Adv_Arr[3] := FALSE;
   S708_TL_DC_U261.Visu_Adv_Arr[4] := FALSE;
   S708_TL_DC_U261.Visu_Adv_Arr[5] := FALSE;
   S708_TL_DC_U261.Visu_Adv_Arr[6] := FALSE;
   S708_TL_DC_U261.Visu_Adv_Arr[7] := FALSE;
   S708_TL_DC_U261.Visu_Adv_Arr[8] := FALSE;
   S708_TL_DC_U261.Visu_Adv_Arr[9] := FALSE;
   S708_TL_DC_U261.Visu_Adv_Arr[10] := FALSE;
   S708_TL_DC_U261.Visu_Adv_Arr[11] := FALSE;
   S708_TL_DC_U261.Visu_Adv_Arr[12] := FALSE;
   S708_TL_DC_U261.Visu_Adv_Arr[13] := FALSE;
   S708_TL_DC_U261.Visu_Adv_Arr[14] := FALSE;
   S708_TL_DC_U261.Visu_Adv_Arr[15] := FALSE;
   S708_TL_DC_U261.Visu_Ret_Arr[0] := FALSE;
   S708_TL_DC_U261.Visu_Ret_Arr[1] := FALSE;
   S708_TL_DC_U261.Visu_Ret_Arr[2] := FALSE;
   S708_TL_DC_U261.Visu_Ret_Arr[3] := FALSE;
   S708_TL_DC_U261.Visu_Ret_Arr[4] := FALSE;
   S708_TL_DC_U261.Visu_Ret_Arr[5] := FALSE;
   S708_TL_DC_U261.Visu_Ret_Arr[6] := FALSE;
   S708_TL_DC_U261.Visu_Ret_Arr[7] := FALSE;
   S708_TL_DC_U261.Visu_Ret_Arr[8] := FALSE;
   S708_TL_DC_U261.Visu_Ret_Arr[9] := FALSE;
   S708_TL_DC_U261.Visu_Ret_Arr[10] := FALSE;
   S708_TL_DC_U261.Visu_Ret_Arr[11] := FALSE;
   S708_TL_DC_U261.Visu_Ret_Arr[12] := FALSE;
   S708_TL_DC_U261.Visu_Ret_Arr[13] := FALSE;
   S708_TL_DC_U261.Visu_Ret_Arr[14] := FALSE;
   S708_TL_DC_U261.Visu_Ret_Arr[15] := FALSE;
   S708_TL_DC_U261.BLK_Move_Ret := 0;
   S708_TL_DC_U261.Enable := FALSE;
   S708_TL_DC_U261.Adv_End := FALSE;
   S708_TL_DC_U261.Ret_End := FALSE;
   S708_TL_DC_U261_CLAMP.Enable_Aux := FALSE;
   S708_TL_DC_U261_CLAMP.Adv_Amount := 1;
   S708_TL_DC_U261_CLAMP.Ret_Amount := 1;
   S708_TL_DC_U261_CLAMP.LS_Adv1 := FALSE;
   S708_TL_DC_U261_CLAMP.LS_Ret1 := FALSE;
   S708_TL_DC_U261_CLAMP.LS_Adv2 := FALSE;
   S708_TL_DC_U261_CLAMP.LS_Ret2 := FALSE;
   S708_TL_DC_U261_CLAMP.LS_Adv3 := FALSE;
   S708_TL_DC_U261_CLAMP.LS_Ret3 := FALSE;
   S708_TL_DC_U261_CLAMP.LS_Adv4 := FALSE;
   S708_TL_DC_U261_CLAMP.LS_Ret4 := FALSE;
   S708_TL_DC_U261_CLAMP.LS_Adv5 := FALSE;
   S708_TL_DC_U261_CLAMP.LS_Ret5 := FALSE;
   S708_TL_DC_U261_CLAMP.LS_Adv6 := FALSE;
   S708_TL_DC_U261_CLAMP.LS_Ret6 := FALSE;
   S708_TL_DC_U261_CLAMP.LS_Adv7 := FALSE;
   S708_TL_DC_U261_CLAMP.LS_Ret7 := FALSE;
   S708_TL_DC_U261_CLAMP.LS_Adv8 := FALSE;
   S708_TL_DC_U261_CLAMP.LS_Ret8 := FALSE;
   S708_TL_DC_U261_CLAMP.SOL_Adv := FALSE;
   S708_TL_DC_U261_CLAMP.SOL_Ret := FALSE;
   S708_TL_DC_U261_CLAMP.M_Ready := TRUE;
   S708_TL_DC_U261_CLAMP.T_CHK1 := T#7S;
   S708_TL_DC_U261_CLAMP.T_CHK2 := T#7S;
   S708_TL_DC_U261_CLAMP.PB_Lamp_CHK := FALSE;
   S708_TL_DC_U261_CLAMP.PB_Error_Rst := FALSE;
   S708_TL_DC_U261_CLAMP.M_FLICK := TRUE;
   S708_TL_DC_U261_CLAMP.M_Adv_Err := FALSE;
   S708_TL_DC_U261_CLAMP.M_Ret_Err := FALSE;
   S708_TL_DC_U261_CLAMP.LP_Adv := FALSE;
   S708_TL_DC_U261_CLAMP.LP_Ret := FALSE;
   S708_TL_DC_U261_CLAMP.Visu_Adv := W#16#0;
   S708_TL_DC_U261_CLAMP.Visu_Ret := W#16#0;
   S708_TL_DC_U261_CLAMP.Error_T1.IN := FALSE;
   S708_TL_DC_U261_CLAMP.Error_T1.PT := T#7S;
   S708_TL_DC_U261_CLAMP.Error_T1.Q := FALSE;
   S708_TL_DC_U261_CLAMP.Error_T1.ET := T#0MS;
   S708_TL_DC_U261_CLAMP.Error_T1.STATE := B#16#0;
   S708_TL_DC_U261_CLAMP.Error_T1.STIME := T#23D5H8M48S439MS;
   S708_TL_DC_U261_CLAMP.Error_T1.ATIME := T#23D5H8M49S747MS;
   S708_TL_DC_U261_CLAMP.Error_T2.IN := FALSE;
   S708_TL_DC_U261_CLAMP.Error_T2.PT := T#7S;
   S708_TL_DC_U261_CLAMP.Error_T2.Q := FALSE;
   S708_TL_DC_U261_CLAMP.Error_T2.ET := T#0MS;
   S708_TL_DC_U261_CLAMP.Error_T2.STATE := B#16#0;
   S708_TL_DC_U261_CLAMP.Error_T2.STIME := T#0MS;
   S708_TL_DC_U261_CLAMP.Error_T2.ATIME := T#0MS;
   S708_TL_DC_U261_CLAMP.Adv_End_Aux := FALSE;
   S708_TL_DC_U261_CLAMP.Ret_End_Aux := FALSE;
   S708_TL_DC_U261_CLAMP.CHK_Aux1 := FALSE;
   S708_TL_DC_U261_CLAMP.CHK_Aux2 := FALSE;
   S708_TL_DC_U261_CLAMP.Error_T1_DN := FALSE;
   S708_TL_DC_U261_CLAMP.Error_T2_DN := FALSE;
   S708_TL_DC_U261_CLAMP.Adv_Memo := FALSE;
   S708_TL_DC_U261_CLAMP.Visu_Adv_Arr[0] := FALSE;
   S708_TL_DC_U261_CLAMP.Visu_Adv_Arr[1] := FALSE;
   S708_TL_DC_U261_CLAMP.Visu_Adv_Arr[2] := FALSE;
   S708_TL_DC_U261_CLAMP.Visu_Adv_Arr[3] := FALSE;
   S708_TL_DC_U261_CLAMP.Visu_Adv_Arr[4] := FALSE;
   S708_TL_DC_U261_CLAMP.Visu_Adv_Arr[5] := FALSE;
   S708_TL_DC_U261_CLAMP.Visu_Adv_Arr[6] := FALSE;
   S708_TL_DC_U261_CLAMP.Visu_Adv_Arr[7] := FALSE;
   S708_TL_DC_U261_CLAMP.Visu_Adv_Arr[8] := FALSE;
   S708_TL_DC_U261_CLAMP.Visu_Adv_Arr[9] := FALSE;
   S708_TL_DC_U261_CLAMP.Visu_Adv_Arr[10] := FALSE;
   S708_TL_DC_U261_CLAMP.Visu_Adv_Arr[11] := FALSE;
   S708_TL_DC_U261_CLAMP.Visu_Adv_Arr[12] := FALSE;
   S708_TL_DC_U261_CLAMP.Visu_Adv_Arr[13] := FALSE;
   S708_TL_DC_U261_CLAMP.Visu_Adv_Arr[14] := FALSE;
   S708_TL_DC_U261_CLAMP.Visu_Adv_Arr[15] := FALSE;
   S708_TL_DC_U261_CLAMP.Visu_Ret_Arr[0] := FALSE;
   S708_TL_DC_U261_CLAMP.Visu_Ret_Arr[1] := FALSE;
   S708_TL_DC_U261_CLAMP.Visu_Ret_Arr[2] := FALSE;
   S708_TL_DC_U261_CLAMP.Visu_Ret_Arr[3] := FALSE;
   S708_TL_DC_U261_CLAMP.Visu_Ret_Arr[4] := FALSE;
   S708_TL_DC_U261_CLAMP.Visu_Ret_Arr[5] := FALSE;
   S708_TL_DC_U261_CLAMP.Visu_Ret_Arr[6] := FALSE;
   S708_TL_DC_U261_CLAMP.Visu_Ret_Arr[7] := FALSE;
   S708_TL_DC_U261_CLAMP.Visu_Ret_Arr[8] := FALSE;
   S708_TL_DC_U261_CLAMP.Visu_Ret_Arr[9] := FALSE;
   S708_TL_DC_U261_CLAMP.Visu_Ret_Arr[10] := FALSE;
   S708_TL_DC_U261_CLAMP.Visu_Ret_Arr[11] := FALSE;
   S708_TL_DC_U261_CLAMP.Visu_Ret_Arr[12] := FALSE;
   S708_TL_DC_U261_CLAMP.Visu_Ret_Arr[13] := FALSE;
   S708_TL_DC_U261_CLAMP.Visu_Ret_Arr[14] := FALSE;
   S708_TL_DC_U261_CLAMP.Visu_Ret_Arr[15] := FALSE;
   S708_TL_DC_U261_CLAMP.BLK_Move_Ret := 0;
   S708_TL_DC_U261_CLAMP.Enable := FALSE;
   S708_TL_DC_U261_CLAMP.Adv_End := FALSE;
   S708_TL_DC_U261_CLAMP.Ret_End := FALSE;
   S708_TL_DC_U269.Enable_Aux := FALSE;
   S708_TL_DC_U269.Adv_Amount := 1;
   S708_TL_DC_U269.Ret_Amount := 1;
   S708_TL_DC_U269.LS_Adv1 := FALSE;
   S708_TL_DC_U269.LS_Ret1 := FALSE;
   S708_TL_DC_U269.LS_Adv2 := FALSE;
   S708_TL_DC_U269.LS_Ret2 := FALSE;
   S708_TL_DC_U269.LS_Adv3 := FALSE;
   S708_TL_DC_U269.LS_Ret3 := FALSE;
   S708_TL_DC_U269.LS_Adv4 := FALSE;
   S708_TL_DC_U269.LS_Ret4 := FALSE;
   S708_TL_DC_U269.LS_Adv5 := FALSE;
   S708_TL_DC_U269.LS_Ret5 := FALSE;
   S708_TL_DC_U269.LS_Adv6 := FALSE;
   S708_TL_DC_U269.LS_Ret6 := FALSE;
   S708_TL_DC_U269.LS_Adv7 := FALSE;
   S708_TL_DC_U269.LS_Ret7 := FALSE;
   S708_TL_DC_U269.LS_Adv8 := FALSE;
   S708_TL_DC_U269.LS_Ret8 := FALSE;
   S708_TL_DC_U269.SOL_Adv := FALSE;
   S708_TL_DC_U269.SOL_Ret := FALSE;
   S708_TL_DC_U269.M_Ready := TRUE;
   S708_TL_DC_U269.T_CHK1 := T#4S;
   S708_TL_DC_U269.T_CHK2 := T#4S;
   S708_TL_DC_U269.PB_Lamp_CHK := FALSE;
   S708_TL_DC_U269.PB_Error_Rst := FALSE;
   S708_TL_DC_U269.M_FLICK := TRUE;
   S708_TL_DC_U269.M_Adv_Err := FALSE;
   S708_TL_DC_U269.M_Ret_Err := FALSE;
   S708_TL_DC_U269.LP_Adv := FALSE;
   S708_TL_DC_U269.LP_Ret := FALSE;
   S708_TL_DC_U269.Visu_Adv := W#16#0;
   S708_TL_DC_U269.Visu_Ret := W#16#0;
   S708_TL_DC_U269.Error_T1.IN := FALSE;
   S708_TL_DC_U269.Error_T1.PT := T#4S;
   S708_TL_DC_U269.Error_T1.Q := FALSE;
   S708_TL_DC_U269.Error_T1.ET := T#0MS;
   S708_TL_DC_U269.Error_T1.STATE := B#16#0;
   S708_TL_DC_U269.Error_T1.STIME := T#23D1H32M29S673MS;
   S708_TL_DC_U269.Error_T1.ATIME := T#23D1H32M29S717MS;
   S708_TL_DC_U269.Error_T2.IN := FALSE;
   S708_TL_DC_U269.Error_T2.PT := T#4S;
   S708_TL_DC_U269.Error_T2.Q := FALSE;
   S708_TL_DC_U269.Error_T2.ET := T#0MS;
   S708_TL_DC_U269.Error_T2.STATE := B#16#0;
   S708_TL_DC_U269.Error_T2.STIME := T#0MS;
   S708_TL_DC_U269.Error_T2.ATIME := T#0MS;
   S708_TL_DC_U269.Adv_End_Aux := FALSE;
   S708_TL_DC_U269.Ret_End_Aux := FALSE;
   S708_TL_DC_U269.CHK_Aux1 := FALSE;
   S708_TL_DC_U269.CHK_Aux2 := FALSE;
   S708_TL_DC_U269.Error_T1_DN := FALSE;
   S708_TL_DC_U269.Error_T2_DN := FALSE;
   S708_TL_DC_U269.Adv_Memo := FALSE;
   S708_TL_DC_U269.Visu_Adv_Arr[0] := FALSE;
   S708_TL_DC_U269.Visu_Adv_Arr[1] := FALSE;
   S708_TL_DC_U269.Visu_Adv_Arr[2] := FALSE;
   S708_TL_DC_U269.Visu_Adv_Arr[3] := FALSE;
   S708_TL_DC_U269.Visu_Adv_Arr[4] := FALSE;
   S708_TL_DC_U269.Visu_Adv_Arr[5] := FALSE;
   S708_TL_DC_U269.Visu_Adv_Arr[6] := FALSE;
   S708_TL_DC_U269.Visu_Adv_Arr[7] := FALSE;
   S708_TL_DC_U269.Visu_Adv_Arr[8] := FALSE;
   S708_TL_DC_U269.Visu_Adv_Arr[9] := FALSE;
   S708_TL_DC_U269.Visu_Adv_Arr[10] := FALSE;
   S708_TL_DC_U269.Visu_Adv_Arr[11] := FALSE;
   S708_TL_DC_U269.Visu_Adv_Arr[12] := FALSE;
   S708_TL_DC_U269.Visu_Adv_Arr[13] := FALSE;
   S708_TL_DC_U269.Visu_Adv_Arr[14] := FALSE;
   S708_TL_DC_U269.Visu_Adv_Arr[15] := FALSE;
   S708_TL_DC_U269.Visu_Ret_Arr[0] := FALSE;
   S708_TL_DC_U269.Visu_Ret_Arr[1] := FALSE;
   S708_TL_DC_U269.Visu_Ret_Arr[2] := FALSE;
   S708_TL_DC_U269.Visu_Ret_Arr[3] := FALSE;
   S708_TL_DC_U269.Visu_Ret_Arr[4] := FALSE;
   S708_TL_DC_U269.Visu_Ret_Arr[5] := FALSE;
   S708_TL_DC_U269.Visu_Ret_Arr[6] := FALSE;
   S708_TL_DC_U269.Visu_Ret_Arr[7] := FALSE;
   S708_TL_DC_U269.Visu_Ret_Arr[8] := FALSE;
   S708_TL_DC_U269.Visu_Ret_Arr[9] := FALSE;
   S708_TL_DC_U269.Visu_Ret_Arr[10] := FALSE;
   S708_TL_DC_U269.Visu_Ret_Arr[11] := FALSE;
   S708_TL_DC_U269.Visu_Ret_Arr[12] := FALSE;
   S708_TL_DC_U269.Visu_Ret_Arr[13] := FALSE;
   S708_TL_DC_U269.Visu_Ret_Arr[14] := FALSE;
   S708_TL_DC_U269.Visu_Ret_Arr[15] := FALSE;
   S708_TL_DC_U269.BLK_Move_Ret := 0;
   S708_TL_DC_U269.Enable := FALSE;
   S708_TL_DC_U269.Adv_End := FALSE;
   S708_TL_DC_U269.Ret_End := FALSE;
   S708_TL_DC_U269_CLAMP.Enable_Aux := FALSE;
   S708_TL_DC_U269_CLAMP.Adv_Amount := 1;
   S708_TL_DC_U269_CLAMP.Ret_Amount := 2;
   S708_TL_DC_U269_CLAMP.LS_Adv1 := FALSE;
   S708_TL_DC_U269_CLAMP.LS_Ret1 := FALSE;
   S708_TL_DC_U269_CLAMP.LS_Adv2 := FALSE;
   S708_TL_DC_U269_CLAMP.LS_Ret2 := FALSE;
   S708_TL_DC_U269_CLAMP.LS_Adv3 := FALSE;
   S708_TL_DC_U269_CLAMP.LS_Ret3 := FALSE;
   S708_TL_DC_U269_CLAMP.LS_Adv4 := FALSE;
   S708_TL_DC_U269_CLAMP.LS_Ret4 := FALSE;
   S708_TL_DC_U269_CLAMP.LS_Adv5 := FALSE;
   S708_TL_DC_U269_CLAMP.LS_Ret5 := FALSE;
   S708_TL_DC_U269_CLAMP.LS_Adv6 := FALSE;
   S708_TL_DC_U269_CLAMP.LS_Ret6 := FALSE;
   S708_TL_DC_U269_CLAMP.LS_Adv7 := FALSE;
   S708_TL_DC_U269_CLAMP.LS_Ret7 := FALSE;
   S708_TL_DC_U269_CLAMP.LS_Adv8 := FALSE;
   S708_TL_DC_U269_CLAMP.LS_Ret8 := FALSE;
   S708_TL_DC_U269_CLAMP.SOL_Adv := FALSE;
   S708_TL_DC_U269_CLAMP.SOL_Ret := FALSE;
   S708_TL_DC_U269_CLAMP.M_Ready := TRUE;
   S708_TL_DC_U269_CLAMP.T_CHK1 := T#4S;
   S708_TL_DC_U269_CLAMP.T_CHK2 := T#4S;
   S708_TL_DC_U269_CLAMP.PB_Lamp_CHK := FALSE;
   S708_TL_DC_U269_CLAMP.PB_Error_Rst := FALSE;
   S708_TL_DC_U269_CLAMP.M_FLICK := TRUE;
   S708_TL_DC_U269_CLAMP.M_Adv_Err := FALSE;
   S708_TL_DC_U269_CLAMP.M_Ret_Err := FALSE;
   S708_TL_DC_U269_CLAMP.LP_Adv := FALSE;
   S708_TL_DC_U269_CLAMP.LP_Ret := FALSE;
   S708_TL_DC_U269_CLAMP.Visu_Adv := W#16#0;
   S708_TL_DC_U269_CLAMP.Visu_Ret := W#16#0;
   S708_TL_DC_U269_CLAMP.Error_T1.IN := FALSE;
   S708_TL_DC_U269_CLAMP.Error_T1.PT := T#4S;
   S708_TL_DC_U269_CLAMP.Error_T1.Q := FALSE;
   S708_TL_DC_U269_CLAMP.Error_T1.ET := T#0MS;
   S708_TL_DC_U269_CLAMP.Error_T1.STATE := B#16#0;
   S708_TL_DC_U269_CLAMP.Error_T1.STIME := T#23D5H8M48S439MS;
   S708_TL_DC_U269_CLAMP.Error_T1.ATIME := T#23D5H8M49S101MS;
   S708_TL_DC_U269_CLAMP.Error_T2.IN := FALSE;
   S708_TL_DC_U269_CLAMP.Error_T2.PT := T#4S;
   S708_TL_DC_U269_CLAMP.Error_T2.Q := FALSE;
   S708_TL_DC_U269_CLAMP.Error_T2.ET := T#0MS;
   S708_TL_DC_U269_CLAMP.Error_T2.STATE := B#16#0;
   S708_TL_DC_U269_CLAMP.Error_T2.STIME := T#0MS;
   S708_TL_DC_U269_CLAMP.Error_T2.ATIME := T#0MS;
   S708_TL_DC_U269_CLAMP.Adv_End_Aux := FALSE;
   S708_TL_DC_U269_CLAMP.Ret_End_Aux := FALSE;
   S708_TL_DC_U269_CLAMP.CHK_Aux1 := FALSE;
   S708_TL_DC_U269_CLAMP.CHK_Aux2 := FALSE;
   S708_TL_DC_U269_CLAMP.Error_T1_DN := FALSE;
   S708_TL_DC_U269_CLAMP.Error_T2_DN := FALSE;
   S708_TL_DC_U269_CLAMP.Adv_Memo := FALSE;
   S708_TL_DC_U269_CLAMP.Visu_Adv_Arr[0] := FALSE;
   S708_TL_DC_U269_CLAMP.Visu_Adv_Arr[1] := FALSE;
   S708_TL_DC_U269_CLAMP.Visu_Adv_Arr[2] := FALSE;
   S708_TL_DC_U269_CLAMP.Visu_Adv_Arr[3] := FALSE;
   S708_TL_DC_U269_CLAMP.Visu_Adv_Arr[4] := FALSE;
   S708_TL_DC_U269_CLAMP.Visu_Adv_Arr[5] := FALSE;
   S708_TL_DC_U269_CLAMP.Visu_Adv_Arr[6] := FALSE;
   S708_TL_DC_U269_CLAMP.Visu_Adv_Arr[7] := FALSE;
   S708_TL_DC_U269_CLAMP.Visu_Adv_Arr[8] := FALSE;
   S708_TL_DC_U269_CLAMP.Visu_Adv_Arr[9] := FALSE;
   S708_TL_DC_U269_CLAMP.Visu_Adv_Arr[10] := FALSE;
   S708_TL_DC_U269_CLAMP.Visu_Adv_Arr[11] := FALSE;
   S708_TL_DC_U269_CLAMP.Visu_Adv_Arr[12] := FALSE;
   S708_TL_DC_U269_CLAMP.Visu_Adv_Arr[13] := FALSE;
   S708_TL_DC_U269_CLAMP.Visu_Adv_Arr[14] := FALSE;
   S708_TL_DC_U269_CLAMP.Visu_Adv_Arr[15] := FALSE;
   S708_TL_DC_U269_CLAMP.Visu_Ret_Arr[0] := FALSE;
   S708_TL_DC_U269_CLAMP.Visu_Ret_Arr[1] := FALSE;
   S708_TL_DC_U269_CLAMP.Visu_Ret_Arr[2] := FALSE;
   S708_TL_DC_U269_CLAMP.Visu_Ret_Arr[3] := FALSE;
   S708_TL_DC_U269_CLAMP.Visu_Ret_Arr[4] := FALSE;
   S708_TL_DC_U269_CLAMP.Visu_Ret_Arr[5] := FALSE;
   S708_TL_DC_U269_CLAMP.Visu_Ret_Arr[6] := FALSE;
   S708_TL_DC_U269_CLAMP.Visu_Ret_Arr[7] := FALSE;
   S708_TL_DC_U269_CLAMP.Visu_Ret_Arr[8] := FALSE;
   S708_TL_DC_U269_CLAMP.Visu_Ret_Arr[9] := FALSE;
   S708_TL_DC_U269_CLAMP.Visu_Ret_Arr[10] := FALSE;
   S708_TL_DC_U269_CLAMP.Visu_Ret_Arr[11] := FALSE;
   S708_TL_DC_U269_CLAMP.Visu_Ret_Arr[12] := FALSE;
   S708_TL_DC_U269_CLAMP.Visu_Ret_Arr[13] := FALSE;
   S708_TL_DC_U269_CLAMP.Visu_Ret_Arr[14] := FALSE;
   S708_TL_DC_U269_CLAMP.Visu_Ret_Arr[15] := FALSE;
   S708_TL_DC_U269_CLAMP.BLK_Move_Ret := 0;
   S708_TL_DC_U269_CLAMP.Enable := FALSE;
   S708_TL_DC_U269_CLAMP.Adv_End := FALSE;
   S708_TL_DC_U269_CLAMP.Ret_End := FALSE;
   S708_TL_DC_3RD_CLAMP.Enable_Aux := FALSE;
   S708_TL_DC_3RD_CLAMP.Adv_Amount := 1;
   S708_TL_DC_3RD_CLAMP.Ret_Amount := 1;
   S708_TL_DC_3RD_CLAMP.LS_Adv1 := FALSE;
   S708_TL_DC_3RD_CLAMP.LS_Ret1 := FALSE;
   S708_TL_DC_3RD_CLAMP.LS_Adv2 := FALSE;
   S708_TL_DC_3RD_CLAMP.LS_Ret2 := FALSE;
   S708_TL_DC_3RD_CLAMP.LS_Adv3 := FALSE;
   S708_TL_DC_3RD_CLAMP.LS_Ret3 := FALSE;
   S708_TL_DC_3RD_CLAMP.LS_Adv4 := FALSE;
   S708_TL_DC_3RD_CLAMP.LS_Ret4 := FALSE;
   S708_TL_DC_3RD_CLAMP.LS_Adv5 := FALSE;
   S708_TL_DC_3RD_CLAMP.LS_Ret5 := FALSE;
   S708_TL_DC_3RD_CLAMP.LS_Adv6 := FALSE;
   S708_TL_DC_3RD_CLAMP.LS_Ret6 := FALSE;
   S708_TL_DC_3RD_CLAMP.LS_Adv7 := FALSE;
   S708_TL_DC_3RD_CLAMP.LS_Ret7 := FALSE;
   S708_TL_DC_3RD_CLAMP.LS_Adv8 := FALSE;
   S708_TL_DC_3RD_CLAMP.LS_Ret8 := FALSE;
   S708_TL_DC_3RD_CLAMP.SOL_Adv := FALSE;
   S708_TL_DC_3RD_CLAMP.SOL_Ret := FALSE;
   S708_TL_DC_3RD_CLAMP.M_Ready := TRUE;
   S708_TL_DC_3RD_CLAMP.T_CHK1 := T#4S;
   S708_TL_DC_3RD_CLAMP.T_CHK2 := T#4S;
   S708_TL_DC_3RD_CLAMP.PB_Lamp_CHK := FALSE;
   S708_TL_DC_3RD_CLAMP.PB_Error_Rst := FALSE;
   S708_TL_DC_3RD_CLAMP.M_FLICK := TRUE;
   S708_TL_DC_3RD_CLAMP.M_Adv_Err := FALSE;
   S708_TL_DC_3RD_CLAMP.M_Ret_Err := FALSE;
   S708_TL_DC_3RD_CLAMP.LP_Adv := FALSE;
   S708_TL_DC_3RD_CLAMP.LP_Ret := FALSE;
   S708_TL_DC_3RD_CLAMP.Visu_Adv := W#16#0;
   S708_TL_DC_3RD_CLAMP.Visu_Ret := W#16#0;
   S708_TL_DC_3RD_CLAMP.Error_T1.IN := FALSE;
   S708_TL_DC_3RD_CLAMP.Error_T1.PT := T#4S;
   S708_TL_DC_3RD_CLAMP.Error_T1.Q := FALSE;
   S708_TL_DC_3RD_CLAMP.Error_T1.ET := T#0MS;
   S708_TL_DC_3RD_CLAMP.Error_T1.STATE := B#16#0;
   S708_TL_DC_3RD_CLAMP.Error_T1.STIME := T#23D5H8M46S781MS;
   S708_TL_DC_3RD_CLAMP.Error_T1.ATIME := T#23D5H8M46S825MS;
   S708_TL_DC_3RD_CLAMP.Error_T2.IN := FALSE;
   S708_TL_DC_3RD_CLAMP.Error_T2.PT := T#4S;
   S708_TL_DC_3RD_CLAMP.Error_T2.Q := FALSE;
   S708_TL_DC_3RD_CLAMP.Error_T2.ET := T#0MS;
   S708_TL_DC_3RD_CLAMP.Error_T2.STATE := B#16#0;
   S708_TL_DC_3RD_CLAMP.Error_T2.STIME := T#0MS;
   S708_TL_DC_3RD_CLAMP.Error_T2.ATIME := T#0MS;
   S708_TL_DC_3RD_CLAMP.Adv_End_Aux := FALSE;
   S708_TL_DC_3RD_CLAMP.Ret_End_Aux := FALSE;
   S708_TL_DC_3RD_CLAMP.CHK_Aux1 := FALSE;
   S708_TL_DC_3RD_CLAMP.CHK_Aux2 := FALSE;
   S708_TL_DC_3RD_CLAMP.Error_T1_DN := FALSE;
   S708_TL_DC_3RD_CLAMP.Error_T2_DN := FALSE;
   S708_TL_DC_3RD_CLAMP.Adv_Memo := FALSE;
   S708_TL_DC_3RD_CLAMP.Visu_Adv_Arr[0] := FALSE;
   S708_TL_DC_3RD_CLAMP.Visu_Adv_Arr[1] := FALSE;
   S708_TL_DC_3RD_CLAMP.Visu_Adv_Arr[2] := FALSE;
   S708_TL_DC_3RD_CLAMP.Visu_Adv_Arr[3] := FALSE;
   S708_TL_DC_3RD_CLAMP.Visu_Adv_Arr[4] := FALSE;
   S708_TL_DC_3RD_CLAMP.Visu_Adv_Arr[5] := FALSE;
   S708_TL_DC_3RD_CLAMP.Visu_Adv_Arr[6] := FALSE;
   S708_TL_DC_3RD_CLAMP.Visu_Adv_Arr[7] := FALSE;
   S708_TL_DC_3RD_CLAMP.Visu_Adv_Arr[8] := FALSE;
   S708_TL_DC_3RD_CLAMP.Visu_Adv_Arr[9] := FALSE;
   S708_TL_DC_3RD_CLAMP.Visu_Adv_Arr[10] := FALSE;
   S708_TL_DC_3RD_CLAMP.Visu_Adv_Arr[11] := FALSE;
   S708_TL_DC_3RD_CLAMP.Visu_Adv_Arr[12] := FALSE;
   S708_TL_DC_3RD_CLAMP.Visu_Adv_Arr[13] := FALSE;
   S708_TL_DC_3RD_CLAMP.Visu_Adv_Arr[14] := FALSE;
   S708_TL_DC_3RD_CLAMP.Visu_Adv_Arr[15] := FALSE;
   S708_TL_DC_3RD_CLAMP.Visu_Ret_Arr[0] := FALSE;
   S708_TL_DC_3RD_CLAMP.Visu_Ret_Arr[1] := FALSE;
   S708_TL_DC_3RD_CLAMP.Visu_Ret_Arr[2] := FALSE;
   S708_TL_DC_3RD_CLAMP.Visu_Ret_Arr[3] := FALSE;
   S708_TL_DC_3RD_CLAMP.Visu_Ret_Arr[4] := FALSE;
   S708_TL_DC_3RD_CLAMP.Visu_Ret_Arr[5] := FALSE;
   S708_TL_DC_3RD_CLAMP.Visu_Ret_Arr[6] := FALSE;
   S708_TL_DC_3RD_CLAMP.Visu_Ret_Arr[7] := FALSE;
   S708_TL_DC_3RD_CLAMP.Visu_Ret_Arr[8] := FALSE;
   S708_TL_DC_3RD_CLAMP.Visu_Ret_Arr[9] := FALSE;
   S708_TL_DC_3RD_CLAMP.Visu_Ret_Arr[10] := FALSE;
   S708_TL_DC_3RD_CLAMP.Visu_Ret_Arr[11] := FALSE;
   S708_TL_DC_3RD_CLAMP.Visu_Ret_Arr[12] := FALSE;
   S708_TL_DC_3RD_CLAMP.Visu_Ret_Arr[13] := FALSE;
   S708_TL_DC_3RD_CLAMP.Visu_Ret_Arr[14] := FALSE;
   S708_TL_DC_3RD_CLAMP.Visu_Ret_Arr[15] := FALSE;
   S708_TL_DC_3RD_CLAMP.BLK_Move_Ret := 0;
   S708_TL_DC_3RD_CLAMP.Enable := FALSE;
   S708_TL_DC_3RD_CLAMP.Adv_End := FALSE;
   S708_TL_DC_3RD_CLAMP.Ret_End := FALSE;
   S708_TL_DC_U262_1_UP_DN.Enable_Aux := FALSE;
   S708_TL_DC_U262_1_UP_DN.Adv_Amount := 1;
   S708_TL_DC_U262_1_UP_DN.Ret_Amount := 1;
   S708_TL_DC_U262_1_UP_DN.LS_Adv1 := FALSE;
   S708_TL_DC_U262_1_UP_DN.LS_Ret1 := FALSE;
   S708_TL_DC_U262_1_UP_DN.LS_Adv2 := FALSE;
   S708_TL_DC_U262_1_UP_DN.LS_Ret2 := FALSE;
   S708_TL_DC_U262_1_UP_DN.LS_Adv3 := FALSE;
   S708_TL_DC_U262_1_UP_DN.LS_Ret3 := FALSE;
   S708_TL_DC_U262_1_UP_DN.LS_Adv4 := FALSE;
   S708_TL_DC_U262_1_UP_DN.LS_Ret4 := FALSE;
   S708_TL_DC_U262_1_UP_DN.LS_Adv5 := FALSE;
   S708_TL_DC_U262_1_UP_DN.LS_Ret5 := FALSE;
   S708_TL_DC_U262_1_UP_DN.LS_Adv6 := FALSE;
   S708_TL_DC_U262_1_UP_DN.LS_Ret6 := FALSE;
   S708_TL_DC_U262_1_UP_DN.LS_Adv7 := FALSE;
   S708_TL_DC_U262_1_UP_DN.LS_Ret7 := FALSE;
   S708_TL_DC_U262_1_UP_DN.LS_Adv8 := FALSE;
   S708_TL_DC_U262_1_UP_DN.LS_Ret8 := FALSE;
   S708_TL_DC_U262_1_UP_DN.SOL_Adv := FALSE;
   S708_TL_DC_U262_1_UP_DN.SOL_Ret := FALSE;
   S708_TL_DC_U262_1_UP_DN.M_Ready := TRUE;
   S708_TL_DC_U262_1_UP_DN.T_CHK1 := T#4S;
   S708_TL_DC_U262_1_UP_DN.T_CHK2 := T#4S;
   S708_TL_DC_U262_1_UP_DN.PB_Lamp_CHK := FALSE;
   S708_TL_DC_U262_1_UP_DN.PB_Error_Rst := FALSE;
   S708_TL_DC_U262_1_UP_DN.M_FLICK := TRUE;
   S708_TL_DC_U262_1_UP_DN.M_Adv_Err := FALSE;
   S708_TL_DC_U262_1_UP_DN.M_Ret_Err := FALSE;
   S708_TL_DC_U262_1_UP_DN.LP_Adv := FALSE;
   S708_TL_DC_U262_1_UP_DN.LP_Ret := FALSE;
   S708_TL_DC_U262_1_UP_DN.Visu_Adv := W#16#0;
   S708_TL_DC_U262_1_UP_DN.Visu_Ret := W#16#0;
   S708_TL_DC_U262_1_UP_DN.Error_T1.IN := FALSE;
   S708_TL_DC_U262_1_UP_DN.Error_T1.PT := T#4S;
   S708_TL_DC_U262_1_UP_DN.Error_T1.Q := FALSE;
   S708_TL_DC_U262_1_UP_DN.Error_T1.ET := T#0MS;
